    |   movel([0.647232, -1.413618, -2.553262, -0.745508, 1.570796, 2.218028],accel_mss,speed_ms,0,blend_radius_m)
    |   movel([0.645203, -1.414719, -2.552433, -0.745237, 1.570796, 2.216000],accel_mss,speed_ms,0,blend_radius_m)
    |   speed_ms = 0.005
    |   movel([0.645203, -1.406157, -2.548592, -0.757639, 1.570796, 2.216000],accel_mss,speed_ms,0,blend_radius_m)
    |   speed_ms = 0.040
    |   movel([0.644708, -1.402598, -2.551232, -0.758559, 1.570796, 2.215504],accel_mss,speed_ms,0,blend_radius_m)
    |   speed_ms = 0.005
    |   movel([0.644708, -1.411187, -2.555088, -0.746114, 1.570796, 2.215504],accel_mss,speed_ms,0,blend_radius_m)
    |   speed_ms = 0.025
    |   movel([0.632928, -1.420166, -2.548302, -0.743920, 1.570796, 2.203724],accel_mss,speed_ms,0,blend_radius_m)
    |   movel([0.632254, -1.420811, -2.547810, -0.743767, 1.570796, 2.203050],accel_mss,speed_ms,0,blend_radius_m)
    |   movel([0.631894, -1.421742, -2.547099, -0.743548, 1.570796, 2.202690],accel_mss,speed_ms,0,blend_radius_m)
    |   movel([0.631428, -1.422941, -2.546181, -0.743267, 1.570796, 2.202224],accel_mss,speed_ms,0,blend_radius_m)
    |   movel([0.630697, -1.424121, -2.545275, -0.742992, 1.570796, 2.201494],accel_mss,speed_ms,0,blend_radius_m)
    |   speed_ms = 0.005
    |   movel([0.630697, -1.415631, -2.541475, -0.755283, 1.570796, 2.201494],accel_mss,speed_ms,0,blend_radius_m)
    |   speed_ms = 0.040
    |   movel([0.643692, -1.414403, -2.542405, -0.755581, 1.570796, 2.214488],accel_mss,speed_ms,0,blend_radius_m)
    |   speed_ms = 0.005
    |   movel([0.643692, -1.422902, -2.546211, -0.743276, 1.570796, 2.214488],accel_mss,speed_ms,0,blend_radius_m)
    |   speed_ms = 0.025
    |   movel([0.644486, -1.421667, -2.547157, -0.743566, 1.570796, 2.215283],accel_mss,speed_ms,0,blend_radius_m)
    |   movel([0.645426, -1.420470, -2.548071, -0.743848, 1.570796, 2.216222],accel_mss,speed_ms,0,blend_radius_m)
    |   movel([0.646493, -1.419333, -2.548937, -0.744119, 1.570796, 2.217289],accel_mss,speed_ms,0,blend_radius_m)
    |   movel([0.647675, -1.418273, -2.549743, -0.744373, 1.570796, 2.218471],accel_mss,speed_ms,0,blend_radius_m)
    |   movel([0.648555, -1.417600, -2.550254, -0.744535, 1.570796, 2.219351],accel_mss,speed_ms,0,blend_radius_m)
    |   movel([0.649486, -1.417003, -2.550706, -0.744680, 1.570796, 2.220283],accel_mss,speed_ms,0,blend_radius_m)
    |   movel([0.650446, -1.416529, -2.551066, -0.744795, 1.570796, 2.221242],accel_mss,speed_ms,0,blend_radius_m)
    |   movel([0.651421, -1.416216, -2.551302, -0.744871, 1.570796, 2.222217],accel_mss,speed_ms,0,blend_radius_m)
    |   movel([0.652201, -1.416139, -2.551360, -0.744889, 1.570796, 2.222997],accel_mss,speed_ms,0,blend_radius_m)
    |   movel([0.652960, -1.416240, -2.551284, -0.744865, 1.570796, 2.223756],accel_mss,speed_ms,0,blend_radius_m)
    |   movel([0.653689, -1.416481, -2.551102, -0.744806, 1.570796, 2.224486],accel_mss,speed_ms,0,blend_radius_m)
    |   movel([0.654385, -1.416828, -2.550839, -0.744722, 1.570796, 2.225181],accel_mss,speed_ms,0,blend_radius_m)
    |   movel([0.655645, -1.417690, -2.550186, -0.744513, 1.570796, 2.226441],accel_mss,speed_ms,0,blend_radius_m)
    |   movel([0.656685, -1.418543, -2.549538, -0.744308, 1.570796, 2.227481],accel_mss,speed_ms,0,blend_radius_m)
    |   movel([0.655905, -1.418044, -2.549917, -0.744428, 1.570796, 2.226701],accel_mss,speed_ms,0,blend_radius_m)
    |   movel([0.654985, -1.417739, -2.550148, -0.744502, 1.570796, 2.225782],accel_mss,speed_ms,0,blend_radius_m)
    |   movel([0.653930, -1.417662, -2.550207, -0.744520, 1.570796, 2.224726],accel_mss,speed_ms,0,blend_radius_m)
    |   movel([0.652738, -1.417850, -2.550064, -0.744475, 1.570796, 2.223534],accel_mss,speed_ms,0,blend_radius_m)
    |   movel([0.651666, -1.418237, -2.549770, -0.744382, 1.570796, 2.222463],accel_mss,speed_ms,0,blend_radius_m)
    |   movel([0.650613, -1.418779, -2.549358, -0.744251, 1.570796, 2.221410],accel_mss,speed_ms,0,blend_radius_m)
    |   movel([0.649643, -1.419392, -2.548892, -0.744105, 1.570796, 2.220440],accel_mss,speed_ms,0,blend_radius_m)
    |   movel([0.648729, -1.420086, -2.548363, -0.743939, 1.570796, 2.219525],accel_mss,speed_ms,0,blend_radius_m)
    |   movel([0.647076, -1.421670, -2.547154, -0.743565, 1.570796, 2.217872],accel_mss,speed_ms,0,blend_radius_m)
    |   movel([0.645680, -1.423421, -2.545813, -0.743155, 1.570796, 2.216476],accel_mss,speed_ms,0,blend_radius_m)
    |   movel([0.644476, -1.425396, -2.544295, -0.742698, 1.570796, 2.215272],accel_mss,speed_ms,0,blend_radius_m)
    |   speed_ms = 0.005
    |   movel([0.644476, -1.416915, -2.540500, -0.754974, 1.570796, 2.215272],accel_mss,speed_ms,0,blend_radius_m)
    |   speed_ms = 0.040
    |   movel([0.649184, -1.413818, -2.542847, -0.755724, 1.570796, 2.219981],accel_mss,speed_ms,0,blend_radius_m)
    |   speed_ms = 0.005
    |   movel([0.649184, -1.422322, -2.546655, -0.743412, 1.570796, 2.219981],accel_mss,speed_ms,0,blend_radius_m)
    |   speed_ms = 0.025
    |   movel([0.648903, -1.422543, -2.546486, -0.743360, 1.570796, 2.219700],accel_mss,speed_ms,0,blend_radius_m)
    |   movel([0.648598, -1.422527, -2.546498, -0.743364, 1.570796, 2.219395],accel_mss,speed_ms,0,blend_radius_m)
    |   movel([0.648528, -1.422285, -2.546684, -0.743420, 1.570796, 2.219324],accel_mss,speed_ms,0,blend_radius_m)
    |   movel([0.648665, -1.421972, -2.546923, -0.743494, 1.570796, 2.219461],accel_mss,speed_ms,0,blend_radius_m)
    |   movel([0.649263, -1.421482, -2.547298, -0.743609, 1.570796, 2.220060],accel_mss,speed_ms,0,blend_radius_m)
    |   movel([0.649575, -1.421351, -2.547398, -0.743640, 1.570796, 2.220372],accel_mss,speed_ms,0,blend_radius_m)
    |   movel([0.649805, -1.421455, -2.547318, -0.743615, 1.570796, 2.220601],accel_mss,speed_ms,0,blend_radius_m)
    |   movel([0.649814, -1.421733, -2.547106, -0.743550, 1.570796, 2.220610],accel_mss,speed_ms,0,blend_radius_m)
    |   movel([0.649380, -1.422307, -2.546666, -0.743415, 1.570796, 2.220177],accel_mss,speed_ms,0,blend_radius_m)
    |   speed_ms = 0.005
    |   movel([0.649380, -1.413803, -2.542859, -0.755727, 1.570796, 2.220177],accel_mss,speed_ms,0,blend_radius_m)
    |   speed_ms = 0.040
    |   movel([0.644877, -1.421865, -2.536719, -0.753805, 1.570796, 2.215673],accel_mss,speed_ms,0,blend_radius_m)
    |   speed_ms = 0.005
    |   movel([0.644877, -1.430308, -2.540493, -0.741588, 1.570796, 2.215673],accel_mss,speed_ms,0,blend_radius_m)
    |   speed_ms = 0.025
    |   movel([0.646228, -1.429676, -2.540984, -0.741729, 1.570796, 2.217025],accel_mss,speed_ms,0,blend_radius_m)
    |   movel([0.647479, -1.428899, -2.541587, -0.741903, 1.570796, 2.218275],accel_mss,speed_ms,0,blend_radius_m)
    |   movel([0.649990, -1.427329, -2.542803, -0.742257, 1.570796, 2.220786],accel_mss,speed_ms,0,blend_radius_m)
    |   movel([0.651879, -1.426482, -2.543457, -0.742450, 1.570796, 2.222676],accel_mss,speed_ms,0,blend_radius_m)
    |   movel([0.657788, -1.424441, -2.545030, -0.742919, 1.570796, 2.228584],accel_mss,speed_ms,0,blend_radius_m)
    |   movel([0.658989, -1.423871, -2.545467, -0.743050, 1.570796, 2.229786],accel_mss,speed_ms,0,blend_radius_m)
    |   movel([0.659479, -1.423475, -2.545772, -0.743143, 1.570796, 2.230276],accel_mss,speed_ms,0,blend_radius_m)
    |   movel([0.659777, -1.422996, -2.546139, -0.743254, 1.570796, 2.230574],accel_mss,speed_ms,0,blend_radius_m)
    |   movel([0.659769, -1.422425, -2.546576, -0.743387, 1.570796, 2.230566],accel_mss,speed_ms,0,blend_radius_m)
    |   movel([0.659492, -1.421965, -2.546929, -0.743495, 1.570796, 2.230288],accel_mss,speed_ms,0,blend_radius_m)
    |   movel([0.658947, -1.421394, -2.547365, -0.743630, 1.570796, 2.229744],accel_mss,speed_ms,0,blend_radius_m)
    |   movel([0.658295, -1.421032, -2.547641, -0.743715, 1.570796, 2.229091],accel_mss,speed_ms,0,blend_radius_m)
    |   movel([0.657480, -1.420873, -2.547763, -0.743753, 1.570796, 2.228276],accel_mss,speed_ms,0,blend_radius_m)
    |   movel([0.656449, -1.420910, -2.547735, -0.743744, 1.570796, 2.227245],accel_mss,speed_ms,0,blend_radius_m)
    |   movel([0.655264, -1.421153, -2.547549, -0.743687, 1.570796, 2.226060],accel_mss,speed_ms,0,blend_radius_m)
    |   movel([0.654014, -1.421592, -2.547214, -0.743583, 1.570796, 2.224810],accel_mss,speed_ms,0,blend_radius_m)
    |   movel([0.652729, -1.422184, -2.546761, -0.743444, 1.570796, 2.223525],accel_mss,speed_ms,0,blend_radius_m)
    |   movel([0.651431, -1.422893, -2.546218, -0.743278, 1.570796, 2.222227],accel_mss,speed_ms,0,blend_radius_m)
    |   movel([0.648915, -1.424490, -2.544992, -0.742907, 1.570796, 2.219711],accel_mss,speed_ms,0,blend_radius_m)
    |   movel([0.646678, -1.426064, -2.543780, -0.742545, 1.570796, 2.217474],accel_mss,speed_ms,0,blend_radius_m)
    |   movel([0.642614, -1.429086, -2.541442, -0.741861, 1.570796, 2.213410],accel_mss,speed_ms,0,blend_radius_m)
    |   movel([0.641217, -1.430012, -2.540723, -0.741654, 1.570796, 2.212013],accel_mss,speed_ms,0,blend_radius_m)
    |   movel([0.639755, -1.430829, -2.540087, -0.741473, 1.570796, 2.210551],accel_mss,speed_ms,0,blend_radius_m)
    |   movel([0.638252, -1.431473, -2.539586, -0.741330, 1.570796, 2.209049],accel_mss,speed_ms,0,blend_radius_m)
    |   movel([0.636769, -1.431875, -2.539272, -0.741242, 1.570796, 2.207566],accel_mss,speed_ms,0,blend_radius_m)
    |   movel([0.635365, -1.431969, -2.539199, -0.741221, 1.570796, 2.206162],accel_mss,speed_ms,0,blend_radius_m)
    |   movel([0.636219, -1.432324, -2.538922, -0.741143, 1.570796, 2.207016],accel_mss,speed_ms,0,blend_radius_m)
    |   movel([0.637153, -1.432573, -2.538727, -0.741089, 1.570796, 2.207950],accel_mss,speed_ms,0,blend_radius_m)
    |   movel([0.638159, -1.432712, -2.538619, -0.741058, 1.570796, 2.208955],accel_mss,speed_ms,0,blend_radius_m)
    |   movel([0.639218, -1.432740, -2.538596, -0.741052, 1.570796, 2.210014],accel_mss,speed_ms,0,blend_radius_m)
    |   movel([0.638520, -1.433919, -2.537675, -0.740796, 1.570796, 2.209316],accel_mss,speed_ms,0,blend_radius_m)
    |   movel([0.637653, -1.435054, -2.536785, -0.740551, 1.570796, 2.208449],accel_mss,speed_ms,0,blend_radius_m)
    |   movel([0.636642, -1.436119, -2.535948, -0.740322, 1.570796, 2.207438],accel_mss,speed_ms,0,blend_radius_m)
    |   movel([0.635508, -1.437089, -2.535184, -0.740116, 1.570796, 2.206304],accel_mss,speed_ms,0,blend_radius_m)
    |   movel([0.637021, -1.436449, -2.535688, -0.740252, 1.570796, 2.207818],accel_mss,speed_ms,0,blend_radius_m)
    |   movel([0.638475, -1.435651, -2.536316, -0.740422, 1.570796, 2.209271],accel_mss,speed_ms,0,blend_radius_m)
    |   movel([0.639868, -1.434716, -2.537050, -0.740623, 1.570796, 2.210664],accel_mss,speed_ms,0,blend_radius_m)
    |   movel([0.641204, -1.433667, -2.537872, -0.740850, 1.570796, 2.212000],accel_mss,speed_ms,0,blend_radius_m)
    |   movel([0.640775, -1.434467, -2.537245, -0.740677, 1.570796, 2.211571],accel_mss,speed_ms,0,blend_radius_m)
    |   movel([0.640145, -1.435303, -2.536589, -0.740497, 1.570796, 2.210942],accel_mss,speed_ms,0,blend_radius_m)
    |   movel([0.636793, -1.438812, -2.533824, -0.739753, 1.570796, 2.207590],accel_mss,speed_ms,0,blend_radius_m)
    |   movel([0.636040, -1.439697, -2.533123, -0.739568, 1.570796, 2.206837],accel_mss,speed_ms,0,blend_radius_m)
    |   movel([0.635442, -1.440567, -2.532434, -0.739388, 1.570796, 2.206238],accel_mss,speed_ms,0,blend_radius_m)
    |   movel([0.636724, -1.439441, -2.533327, -0.739622, 1.570796, 2.207520],accel_mss,speed_ms,0,blend_radius_m)
    |   movel([0.638005, -1.438470, -2.534094, -0.739825, 1.570796, 2.208801],accel_mss,speed_ms,0,blend_radius_m)
    |   movel([0.640578, -1.436842, -2.535379, -0.740168, 1.570796, 2.211374],accel_mss,speed_ms,0,blend_radius_m)
    |   movel([0.643201, -1.435348, -2.536554, -0.740487, 1.570796, 2.213998],accel_mss,speed_ms,0,blend_radius_m)
    |   movel([0.645926, -1.433653, -2.537883, -0.740853, 1.570796, 2.216722],accel_mss,speed_ms,0,blend_radius_m)
    |   movel([0.647510, -1.432448, -2.538825, -0.741116, 1.570796, 2.218306],accel_mss,speed_ms,0,blend_radius_m)
    |   movel([0.648453, -1.431852, -2.539290, -0.741247, 1.570796, 2.219250],accel_mss,speed_ms,0,blend_radius_m)
    |   movel([0.648851, -1.431691, -2.539416, -0.741282, 1.570796, 2.219647],accel_mss,speed_ms,0,blend_radius_m)
    |   movel([0.649160, -1.431671, -2.539432, -0.741287, 1.570796, 2.219957],accel_mss,speed_ms,0,blend_radius_m)
    |   movel([0.649355, -1.431804, -2.539328, -0.741258, 1.570796, 2.220151],accel_mss,speed_ms,0,blend_radius_m)
    |   movel([0.649443, -1.432056, -2.539131, -0.741202, 1.570796, 2.220239],accel_mss,speed_ms,0,blend_radius_m)
    |   movel([0.649367, -1.432776, -2.538568, -0.741044, 1.570796, 2.220164],accel_mss,speed_ms,0,blend_radius_m)
    |   movel([0.649054, -1.433558, -2.537957, -0.740874, 1.570796, 2.219850],accel_mss,speed_ms,0,blend_radius_m)
    |   movel([0.648620, -1.434127, -2.537512, -0.740751, 1.570796, 2.219417],accel_mss,speed_ms,0,blend_radius_m)
    |   movel([0.650492, -1.432463, -2.538813, -0.741113, 1.570796, 2.221288],accel_mss,speed_ms,0,blend_radius_m)
    |   movel([0.652210, -1.430675, -2.540207, -0.741507, 1.570796, 2.223006],accel_mss,speed_ms,0,blend_radius_m)
    |   movel([0.653753, -1.428790, -2.541671, -0.741927, 1.570796, 2.224549],accel_mss,speed_ms,0,blend_radius_m)
    |   movel([0.655098, -1.426832, -2.543187, -0.742370, 1.570796, 2.225894],accel_mss,speed_ms,0,blend_radius_m)
    |   speed_ms = 0.005
    |   movel([0.655098, -1.418363, -2.539398, -0.754628, 1.570796, 2.225894],accel_mss,speed_ms,0,blend_radius_m)
    |   speed_ms = 0.040
    |   movel([0.656273, -1.420049, -2.538111, -0.754229, 1.570796, 2.227069],accel_mss,speed_ms,0,blend_radius_m)
    |   speed_ms = 0.005
    |   movel([0.656273, -1.428505, -2.541892, -0.741991, 1.570796, 2.227069],accel_mss,speed_ms,0,blend_radius_m)
    |   speed_ms = 0.025
    |   movel([0.657037, -1.429367, -2.541224, -0.741798, 1.570796, 2.227833],accel_mss,speed_ms,0,blend_radius_m)
    |   movel([0.657209, -1.429905, -2.540806, -0.741678, 1.570796, 2.228005],accel_mss,speed_ms,0,blend_radius_m)
    |   movel([0.657126, -1.430531, -2.540319, -0.741539, 1.570796, 2.227923],accel_mss,speed_ms,0,blend_radius_m)
    |   movel([0.656831, -1.431094, -2.539881, -0.741414, 1.570796, 2.227628],accel_mss,speed_ms,0,blend_radius_m)
    |   movel([0.650125, -1.439891, -2.532970, -0.739528, 1.570796, 2.220921],accel_mss,speed_ms,0,blend_radius_m)
    |   movel([0.649615, -1.440501, -2.532486, -0.739402, 1.570796, 2.220412],accel_mss,speed_ms,0,blend_radius_m)
    |   movel([0.649027, -1.441062, -2.532041, -0.739286, 1.570796, 2.219823],accel_mss,speed_ms,0,blend_radius_m)
    |   movel([0.648392, -1.441459, -2.531726, -0.739204, 1.570796, 2.219189],accel_mss,speed_ms,0,blend_radius_m)
    |   movel([0.647752, -1.441583, -2.531627, -0.739179, 1.570796, 2.218548],accel_mss,speed_ms,0,blend_radius_m)
    |   movel([0.647286, -1.441405, -2.531769, -0.739215, 1.570796, 2.218082],accel_mss,speed_ms,0,blend_radius_m)
    |   movel([0.646586, -1.440749, -2.532289, -0.739350, 1.570796, 2.217382],accel_mss,speed_ms,0,blend_radius_m)
    |   movel([0.646108, -1.440597, -2.532410, -0.739382, 1.570796, 2.216904],accel_mss,speed_ms,0,blend_radius_m)
    |   movel([0.645368, -1.440782, -2.532264, -0.739344, 1.570796, 2.216164],accel_mss,speed_ms,0,blend_radius_m)
    |   movel([0.644608, -1.441155, -2.531967, -0.739267, 1.570796, 2.215405],accel_mss,speed_ms,0,blend_radius_m)
    |   movel([0.643699, -1.441518, -2.531678, -0.739192, 1.570796, 2.214496],accel_mss,speed_ms,0,blend_radius_m)
    |   movel([0.642798, -1.441723, -2.531515, -0.739150, 1.570796, 2.213595],accel_mss,speed_ms,0,blend_radius_m)
    |   movel([0.641935, -1.441776, -2.531473, -0.739139, 1.570796, 2.212731],accel_mss,speed_ms,0,blend_radius_m)
    |   movel([0.641134, -1.441682, -2.531548, -0.739159, 1.570796, 2.211931],accel_mss,speed_ms,0,blend_radius_m)
    |   movel([0.640423, -1.441448, -2.531735, -0.739207, 1.570796, 2.211219],accel_mss,speed_ms,0,blend_radius_m)
    |   movel([0.639832, -1.441078, -2.532029, -0.739283, 1.570796, 2.210629],accel_mss,speed_ms,0,blend_radius_m)
    |   movel([0.639385, -1.440582, -2.532422, -0.739385, 1.570796, 2.210182],accel_mss,speed_ms,0,blend_radius_m)
    |   movel([0.639114, -1.439959, -2.532916, -0.739514, 1.570796, 2.209910],accel_mss,speed_ms,0,blend_radius_m)
    |   speed_ms = 0.005
    |   movel([0.639114, -1.431591, -2.529183, -0.751615, 1.570796, 2.209910],accel_mss,speed_ms,0,blend_radius_m)
    |   speed_ms = 0.040
    |   movel([0.629566, -1.437668, -2.524402, -0.750318, 1.570796, 2.200362],accel_mss,speed_ms,0,blend_radius_m)
    |   speed_ms = 0.005
    |   movel([0.629566, -1.445989, -2.528110, -0.738290, 1.570796, 2.200362],accel_mss,speed_ms,0,blend_radius_m)
    |   speed_ms = 0.025
    |   movel([0.624482, -1.455129, -2.520718, -0.736542, 1.570796, 2.195278],accel_mss,speed_ms,0,blend_radius_m)
    |   movel([0.623759, -1.456220, -2.519827, -0.736342, 1.570796, 2.194556],accel_mss,speed_ms,0,blend_radius_m)
    |   movel([0.623285, -1.456679, -2.519452, -0.736258, 1.570796, 2.194081],accel_mss,speed_ms,0,blend_radius_m)
    |   movel([0.622719, -1.457000, -2.519189, -0.736200, 1.570796, 2.193515],accel_mss,speed_ms,0,blend_radius_m)
    |   movel([0.621425, -1.457352, -2.518901, -0.736136, 1.570796, 2.192221],accel_mss,speed_ms,0,blend_radius_m)
    |   movel([0.620864, -1.457799, -2.518534, -0.736056, 1.570796, 2.191661],accel_mss,speed_ms,0,blend_radius_m)
    |   movel([0.620463, -1.458373, -2.518064, -0.735953, 1.570796, 2.191259],accel_mss,speed_ms,0,blend_radius_m)
    |   movel([0.620070, -1.459371, -2.517243, -0.735774, 1.570796, 2.190867],accel_mss,speed_ms,0,blend_radius_m)
    |   movel([0.619927, -1.460382, -2.516412, -0.735596, 1.570796, 2.190723],accel_mss,speed_ms,0,blend_radius_m)
    |   movel([0.619862, -1.462310, -2.514820, -0.735259, 1.570796, 2.190659],accel_mss,speed_ms,0,blend_radius_m)
    |   movel([0.619585, -1.463630, -2.513727, -0.735032, 1.570796, 2.190381],accel_mss,speed_ms,0,blend_radius_m)
    |   movel([0.618938, -1.465519, -2.512159, -0.734712, 1.570796, 2.189734],accel_mss,speed_ms,0,blend_radius_m)
    |   movel([0.618503, -1.466353, -2.511464, -0.734572, 1.570796, 2.189299],accel_mss,speed_ms,0,blend_radius_m)
    |   movel([0.618001, -1.466949, -2.510967, -0.734473, 1.570796, 2.188798],accel_mss,speed_ms,0,blend_radius_m)
    |   movel([0.617730, -1.467114, -2.510829, -0.734446, 1.570796, 2.188526],accel_mss,speed_ms,0,blend_radius_m)
    |   movel([0.617446, -1.467173, -2.510780, -0.734436, 1.570796, 2.188242],accel_mss,speed_ms,0,blend_radius_m)
    |   movel([0.617150, -1.467109, -2.510834, -0.734446, 1.570796, 2.187946],accel_mss,speed_ms,0,blend_radius_m)
    |   movel([0.616845, -1.466904, -2.511005, -0.734480, 1.570796, 2.187641],accel_mss,speed_ms,0,blend_radius_m)
    |   movel([0.616369, -1.467578, -2.510442, -0.734369, 1.570796, 2.187165],accel_mss,speed_ms,0,blend_radius_m)
    |   movel([0.616008, -1.468390, -2.509763, -0.734236, 1.570796, 2.186804],accel_mss,speed_ms,0,blend_radius_m)
    |   movel([0.615555, -1.470239, -2.508214, -0.733936, 1.570796, 2.186351],accel_mss,speed_ms,0,blend_radius_m)
    |   movel([0.615357, -1.472073, -2.506672, -0.733644, 1.570796, 2.186154],accel_mss,speed_ms,0,blend_radius_m)
    |   movel([0.615291, -1.473520, -2.505452, -0.733417, 1.570796, 2.186088],accel_mss,speed_ms,0,blend_radius_m)
    |   movel([0.615441, -1.475063, -2.504147, -0.733179, 1.570796, 2.186237],accel_mss,speed_ms,0,blend_radius_m)
    |   movel([0.615759, -1.476614, -2.502832, -0.732943, 1.570796, 2.186556],accel_mss,speed_ms,0,blend_radius_m)
    |   movel([0.615875, -1.478202, -2.501481, -0.732706, 1.570796, 2.186672],accel_mss,speed_ms,0,blend_radius_m)
    |   movel([0.615743, -1.479016, -2.500787, -0.732586, 1.570796, 2.186540],accel_mss,speed_ms,0,blend_radius_m)
    |   movel([0.615421, -1.479850, -2.500076, -0.732464, 1.570796, 2.186217],accel_mss,speed_ms,0,blend_radius_m)
    |   movel([0.615143, -1.480267, -2.499719, -0.732403, 1.570796, 2.185940],accel_mss,speed_ms,0,blend_radius_m)
    |   movel([0.614767, -1.480641, -2.499399, -0.732349, 1.570796, 2.185563],accel_mss,speed_ms,0,blend_radius_m)
    |   movel([0.614354, -1.480878, -2.499196, -0.732315, 1.570796, 2.185150],accel_mss,speed_ms,0,blend_radius_m)
    |   movel([0.613964, -1.480890, -2.499186, -0.732313, 1.570796, 2.184760],accel_mss,speed_ms,0,blend_radius_m)
    |   movel([0.613760, -1.480715, -2.499336, -0.732338, 1.570796, 2.184557],accel_mss,speed_ms,0,blend_radius_m)
    |   movel([0.613656, -1.480463, -2.499551, -0.732375, 1.570796, 2.184453],accel_mss,speed_ms,0,blend_radius_m)
    |   movel([0.613063, -1.477851, -2.501780, -0.732758, 1.570796, 2.183860],accel_mss,speed_ms,0,blend_radius_m)
    |   movel([0.612918, -1.476478, -2.502947, -0.732964, 1.570796, 2.183714],accel_mss,speed_ms,0,blend_radius_m)
    |   movel([0.612878, -1.475065, -2.504146, -0.733178, 1.570796, 2.183674],accel_mss,speed_ms,0,blend_radius_m)
    |   movel([0.612419, -1.475366, -2.503891, -0.733132, 1.570796, 2.183216],accel_mss,speed_ms,0,blend_radius_m)
    |   movel([0.612028, -1.475740, -2.503573, -0.733075, 1.570796, 2.182824],accel_mss,speed_ms,0,blend_radius_m)
    |   movel([0.611430, -1.476666, -2.502787, -0.732935, 1.570796, 2.182227],accel_mss,speed_ms,0,blend_radius_m)
    |   movel([0.611042, -1.477762, -2.501856, -0.732771, 1.570796, 2.181838],accel_mss,speed_ms,0,blend_radius_m)
    |   movel([0.610826, -1.478948, -2.500845, -0.732596, 1.570796, 2.181622],accel_mss,speed_ms,0,blend_radius_m)
    |   movel([0.610731, -1.481288, -2.498845, -0.732256, 1.570796, 2.181528],accel_mss,speed_ms,0,blend_radius_m)
    |   movel([0.610820, -1.483067, -2.497319, -0.732003, 1.570796, 2.181616],accel_mss,speed_ms,0,blend_radius_m)
    |   movel([0.610778, -1.483746, -2.496735, -0.731908, 1.570796, 2.181574],accel_mss,speed_ms,0,blend_radius_m)
    |   movel([0.610645, -1.484082, -2.496446, -0.731861, 1.570796, 2.181441],accel_mss,speed_ms,0,blend_radius_m)
    |   movel([0.610384, -1.484388, -2.496182, -0.731819, 1.570796, 2.181181],accel_mss,speed_ms,0,blend_radius_m)
    |   movel([0.610011, -1.484627, -2.495976, -0.731786, 1.570796, 2.180807],accel_mss,speed_ms,0,blend_radius_m)
    |   movel([0.609698, -1.484694, -2.495918, -0.731777, 1.570796, 2.180495],accel_mss,speed_ms,0,blend_radius_m)
    |   movel([0.609210, -1.484500, -2.496086, -0.731803, 1.570796, 2.180006],accel_mss,speed_ms,0,blend_radius_m)
    |   movel([0.608588, -1.484138, -2.496398, -0.731854, 1.570796, 2.179384],accel_mss,speed_ms,0,blend_radius_m)
    |   movel([0.608354, -1.484199, -2.496345, -0.731845, 1.570796, 2.179151],accel_mss,speed_ms,0,blend_radius_m)
    |   movel([0.608059, -1.484440, -2.496137, -0.731812, 1.570796, 2.178855],accel_mss,speed_ms,0,blend_radius_m)
    |   movel([0.607831, -1.484776, -2.495847, -0.731765, 1.570796, 2.178627],accel_mss,speed_ms,0,blend_radius_m)
    |   movel([0.607540, -1.485617, -2.495122, -0.731650, 1.570796, 2.178336],accel_mss,speed_ms,0,blend_radius_m)
    |   movel([0.607317, -1.487165, -2.493784, -0.731441, 1.570796, 2.178114],accel_mss,speed_ms,0,blend_radius_m)
    |   movel([0.607067, -1.490393, -2.490980, -0.731016, 1.570796, 2.177864],accel_mss,speed_ms,0,blend_radius_m)
    |   movel([0.606894, -1.493587, -2.488190, -0.730612, 1.570796, 2.177690],accel_mss,speed_ms,0,blend_radius_m)
    |   movel([0.606763, -1.494250, -2.487609, -0.730530, 1.570796, 2.177559],accel_mss,speed_ms,0,blend_radius_m)
    |   movel([0.606487, -1.494923, -2.487018, -0.730448, 1.570796, 2.177283],accel_mss,speed_ms,0,blend_radius_m)
    |   movel([0.606041, -1.495494, -2.486517, -0.730379, 1.570796, 2.176838],accel_mss,speed_ms,0,blend_radius_m)
    |   movel([0.605751, -1.495705, -2.486331, -0.730353, 1.570796, 2.176547],accel_mss,speed_ms,0,blend_radius_m)
    |   movel([0.605086, -1.495899, -2.486161, -0.730330, 1.570796, 2.175882],accel_mss,speed_ms,0,blend_radius_m)
    |   movel([0.604813, -1.495863, -2.486192, -0.730334, 1.570796, 2.175609],accel_mss,speed_ms,0,blend_radius_m)
    |   movel([0.604396, -1.495580, -2.486441, -0.730368, 1.570796, 2.175192],accel_mss,speed_ms,0,blend_radius_m)
    |   movel([0.604131, -1.495116, -2.486849, -0.730424, 1.570796, 2.174927],accel_mss,speed_ms,0,blend_radius_m)
    |   movel([0.603992, -1.494579, -2.487320, -0.730490, 1.570796, 2.174788],accel_mss,speed_ms,0,blend_radius_m)
    |   movel([0.603563, -1.491248, -2.490235, -0.730906, 1.570796, 2.174360],accel_mss,speed_ms,0,blend_radius_m)
    |   movel([0.603337, -1.487825, -2.493211, -0.731352, 1.570796, 2.174133],accel_mss,speed_ms,0,blend_radius_m)
    |   movel([0.603320, -1.484316, -2.496244, -0.731829, 1.570796, 2.174117],accel_mss,speed_ms,0,blend_radius_m)
    |   movel([0.603515, -1.480728, -2.499325, -0.732336, 1.570796, 2.174312],accel_mss,speed_ms,0,blend_radius_m)
    |   movel([0.603673, -1.479373, -2.500483, -0.732533, 1.570796, 2.174470],accel_mss,speed_ms,0,blend_radius_m)
    |   movel([0.604054, -1.477986, -2.501666, -0.732738, 1.570796, 2.174850],accel_mss,speed_ms,0,blend_radius_m)
    |   movel([0.604445, -1.477158, -2.502370, -0.732861, 1.570796, 2.175241],accel_mss,speed_ms,0,blend_radius_m)
    |   movel([0.604935, -1.476340, -2.503064, -0.732984, 1.570796, 2.175732],accel_mss,speed_ms,0,blend_radius_m)
    |   movel([0.606078, -1.474727, -2.504431, -0.733230, 1.570796, 2.176875],accel_mss,speed_ms,0,blend_radius_m)
    |   movel([0.610693, -1.469097, -2.509172, -0.734120, 1.570796, 2.181490],accel_mss,speed_ms,0,blend_radius_m)
    |   movel([0.611871, -1.467453, -2.510546, -0.734389, 1.570796, 2.182668],accel_mss,speed_ms,0,blend_radius_m)
    |   movel([0.612764, -1.465916, -2.511828, -0.734645, 1.570796, 2.183560],accel_mss,speed_ms,0,blend_radius_m)
    |   movel([0.613060, -1.465219, -2.512408, -0.734762, 1.570796, 2.183856],accel_mss,speed_ms,0,blend_radius_m)
    |   movel([0.613226, -1.464587, -2.512933, -0.734869, 1.570796, 2.184023],accel_mss,speed_ms,0,blend_radius_m)
    |   movel([0.613249, -1.464033, -2.513393, -0.734963, 1.570796, 2.184045],accel_mss,speed_ms,0,blend_radius_m)
    |   movel([0.613109, -1.463570, -2.513777, -0.735042, 1.570796, 2.183906],accel_mss,speed_ms,0,blend_radius_m)
    |   movel([0.612615, -1.462930, -2.514307, -0.735152, 1.570796, 2.183411],accel_mss,speed_ms,0,blend_radius_m)
    |   movel([0.612428, -1.462587, -2.514591, -0.735211, 1.570796, 2.183224],accel_mss,speed_ms,0,blend_radius_m)
    |   movel([0.612411, -1.462174, -2.514932, -0.735283, 1.570796, 2.183207],accel_mss,speed_ms,0,blend_radius_m)
    |   movel([0.612772, -1.461510, -2.515481, -0.735398, 1.570796, 2.183569],accel_mss,speed_ms,0,blend_radius_m)
    |   movel([0.613381, -1.460896, -2.515988, -0.735505, 1.570796, 2.184177],accel_mss,speed_ms,0,blend_radius_m)
    |   movel([0.615399, -1.458974, -2.517570, -0.735845, 1.570796, 2.186195],accel_mss,speed_ms,0,blend_radius_m)
    |   movel([0.617306, -1.456995, -2.519193, -0.736201, 1.570796, 2.188103],accel_mss,speed_ms,0,blend_radius_m)
    |   movel([0.619122, -1.454960, -2.520856, -0.736573, 1.570796, 2.189918],accel_mss,speed_ms,0,blend_radius_m)
    |   movel([0.620860, -1.452875, -2.522553, -0.736961, 1.570796, 2.191657],accel_mss,speed_ms,0,blend_radius_m)
    |   movel([0.624183, -1.448586, -2.526023, -0.737780, 1.570796, 2.194980],accel_mss,speed_ms,0,blend_radius_m)
    |   movel([0.627417, -1.444166, -2.529568, -0.738654, 1.570796, 2.198213],accel_mss,speed_ms,0,blend_radius_m)
    |   speed_ms = 0.005
    |   movel([0.627417, -1.435831, -2.525853, -0.750704, 1.570796, 2.198213],accel_mss,speed_ms,0,blend_radius_m)
    |   speed_ms = 0.040
    |   movel([0.617703, -1.446063, -2.517707, -0.748620, 1.570796, 2.188499],accel_mss,speed_ms,0,blend_radius_m)
    |   speed_ms = 0.005
    |   movel([0.617703, -1.454317, -2.521380, -0.736692, 1.570796, 2.188499],accel_mss,speed_ms,0,blend_radius_m)
    |   speed_ms = 0.025
    |   movel([0.614220, -1.456040, -2.519974, -0.736375, 1.570796, 2.185017],accel_mss,speed_ms,0,blend_radius_m)
    |   movel([0.610716, -1.457622, -2.518679, -0.736087, 1.570796, 2.181513],accel_mss,speed_ms,0,blend_radius_m)
    |   movel([0.607196, -1.459065, -2.517495, -0.735829, 1.570796, 2.177992],accel_mss,speed_ms,0,blend_radius_m)
    |   movel([0.603671, -1.460362, -2.516428, -0.735599, 1.570796, 2.174468],accel_mss,speed_ms,0,blend_radius_m)
    |   movel([0.606791, -1.458463, -2.517990, -0.735936, 1.570796, 2.177587],accel_mss,speed_ms,0,blend_radius_m)
    |   movel([0.609822, -1.456386, -2.519691, -0.736312, 1.570796, 2.180619],accel_mss,speed_ms,0,blend_radius_m)
    |   movel([0.612746, -1.454144, -2.521521, -0.736724, 1.570796, 2.183542],accel_mss,speed_ms,0,blend_radius_m)
    |   movel([0.615543, -1.451749, -2.523466, -0.737173, 1.570796, 2.186340],accel_mss,speed_ms,0,blend_radius_m)
    |   movel([0.612639, -1.453118, -2.522356, -0.736916, 1.570796, 2.183435],accel_mss,speed_ms,0,blend_radius_m)
    |   movel([0.609722, -1.454378, -2.521330, -0.736681, 1.570796, 2.180518],accel_mss,speed_ms,0,blend_radius_m)
    |   movel([0.606793, -1.455529, -2.520391, -0.736468, 1.570796, 2.177589],accel_mss,speed_ms,0,blend_radius_m)
    |   movel([0.603861, -1.456566, -2.519544, -0.736279, 1.570796, 2.174657],accel_mss,speed_ms,0,blend_radius_m)
    |   movel([0.600601, -1.457644, -2.518662, -0.736084, 1.570796, 2.171397],accel_mss,speed_ms,0,blend_radius_m)
    |   movel([0.597364, -1.458897, -2.517633, -0.735859, 1.570796, 2.168160],accel_mss,speed_ms,0,blend_radius_m)
    |   movel([0.595768, -1.459689, -2.516982, -0.735718, 1.570796, 2.166565],accel_mss,speed_ms,0,blend_radius_m)
    |   movel([0.594229, -1.460623, -2.516212, -0.735553, 1.570796, 2.165025],accel_mss,speed_ms,0,blend_radius_m)
    |   movel([0.592805, -1.461704, -2.515321, -0.735364, 1.570796, 2.163602],accel_mss,speed_ms,0,blend_radius_m)
    |   movel([0.591552, -1.462929, -2.514307, -0.735152, 1.570796, 2.162348],accel_mss,speed_ms,0,blend_radius_m)
    |   movel([0.592804, -1.461262, -2.515686, -0.735441, 1.570796, 2.163600],accel_mss,speed_ms,0,blend_radius_m)
    |   movel([0.594211, -1.459598, -2.517057, -0.735734, 1.570796, 2.165007],accel_mss,speed_ms,0,blend_radius_m)
    |   movel([0.595752, -1.457957, -2.518405, -0.736027, 1.570796, 2.166548],accel_mss,speed_ms,0,blend_radius_m)
    |   movel([0.597405, -1.456357, -2.519715, -0.736317, 1.570796, 2.168201],accel_mss,speed_ms,0,blend_radius_m)
    |   movel([0.599146, -1.454818, -2.520971, -0.736599, 1.570796, 2.169942],accel_mss,speed_ms,0,blend_radius_m)
    |   movel([0.600954, -1.453361, -2.522158, -0.736870, 1.570796, 2.171750],accel_mss,speed_ms,0,blend_radius_m)
    |   movel([0.602805, -1.452004, -2.523260, -0.737125, 1.570796, 2.173601],accel_mss,speed_ms,0,blend_radius_m)
    |   movel([0.604675, -1.450769, -2.524260, -0.737360, 1.570796, 2.175471],accel_mss,speed_ms,0,blend_radius_m)
    |   movel([0.601533, -1.452451, -2.522897, -0.737041, 1.570796, 2.172329],accel_mss,speed_ms,0,blend_radius_m)
    |   movel([0.598460, -1.454267, -2.521421, -0.736701, 1.570796, 2.169257],accel_mss,speed_ms,0,blend_radius_m)
    |   movel([0.595458, -1.456198, -2.519845, -0.736346, 1.570796, 2.166254],accel_mss,speed_ms,0,blend_radius_m)
    |   movel([0.592526, -1.458228, -2.518182, -0.735978, 1.570796, 2.163322],accel_mss,speed_ms,0,blend_radius_m)
    |   movel([0.589668, -1.460337, -2.516448, -0.735603, 1.570796, 2.160464],accel_mss,speed_ms,0,blend_radius_m)
    |   movel([0.586882, -1.462508, -2.514656, -0.735225, 1.570796, 2.157678],accel_mss,speed_ms,0,blend_radius_m)
    |   movel([0.581527, -1.466961, -2.510957, -0.734471, 1.570796, 2.152324],accel_mss,speed_ms,0,blend_radius_m)
    |   movel([0.583200, -1.465285, -2.512353, -0.734751, 1.570796, 2.153996],accel_mss,speed_ms,0,blend_radius_m)
    |   movel([0.584790, -1.463356, -2.513954, -0.735079, 1.570796, 2.155586],accel_mss,speed_ms,0,blend_radius_m)
    |   movel([0.587772, -1.459527, -2.517115, -0.735747, 1.570796, 2.158569],accel_mss,speed_ms,0,blend_radius_m)
    |   movel([0.589223, -1.457899, -2.518453, -0.736038, 1.570796, 2.160019],accel_mss,speed_ms,0,blend_radius_m)
    |   movel([0.590627, -1.456498, -2.519600, -0.736291, 1.570796, 2.161423],accel_mss,speed_ms,0,blend_radius_m)
    |   movel([0.593740, -1.453771, -2.521825, -0.736794, 1.570796, 2.164536],accel_mss,speed_ms,0,blend_radius_m)
    |   movel([0.593201, -1.454066, -2.521585, -0.736739, 1.570796, 2.163998],accel_mss,speed_ms,0,blend_radius_m)
    |   movel([0.592392, -1.454326, -2.521373, -0.736690, 1.570796, 2.163188],accel_mss,speed_ms,0,blend_radius_m)
    |   movel([0.588113, -1.455156, -2.520696, -0.736537, 1.570796, 2.158910],accel_mss,speed_ms,0,blend_radius_m)
    |   movel([0.586531, -1.455538, -2.520385, -0.736467, 1.570796, 2.157327],accel_mss,speed_ms,0,blend_radius_m)
    |   movel([0.584569, -1.456412, -2.519671, -0.736307, 1.570796, 2.155365],accel_mss,speed_ms,0,blend_radius_m)
    |   movel([0.582619, -1.457507, -2.518774, -0.736108, 1.570796, 2.153415],accel_mss,speed_ms,0,blend_radius_m)
    |   movel([0.578875, -1.459968, -2.516752, -0.735669, 1.570796, 2.149671],accel_mss,speed_ms,0,blend_radius_m)
    |   movel([0.580598, -1.458430, -2.518017, -0.735942, 1.570796, 2.151394],accel_mss,speed_ms,0,blend_radius_m)
    |   movel([0.582217, -1.456797, -2.519355, -0.736237, 1.570796, 2.153013],accel_mss,speed_ms,0,blend_radius_m)
    |   movel([0.585431, -1.453485, -2.522057, -0.736847, 1.570796, 2.156227],accel_mss,speed_ms,0,blend_radius_m)
    |   movel([0.587232, -1.451864, -2.523373, -0.737152, 1.570796, 2.158029],accel_mss,speed_ms,0,blend_radius_m)
    |   movel([0.589151, -1.450323, -2.524621, -0.737445, 1.570796, 2.159948],accel_mss,speed_ms,0,blend_radius_m)
    |   movel([0.593248, -1.447424, -2.526958, -0.738007, 1.570796, 2.164045],accel_mss,speed_ms,0,blend_radius_m)
    |   movel([0.601686, -1.442016, -2.531283, -0.739090, 1.570796, 2.172482],accel_mss,speed_ms,0,blend_radius_m)
    |   movel([0.599268, -1.442212, -2.531127, -0.739050, 1.570796, 2.170065],accel_mss,speed_ms,0,blend_radius_m)
    |   movel([0.596800, -1.442588, -2.530827, -0.738974, 1.570796, 2.167597],accel_mss,speed_ms,0,blend_radius_m)
    |   movel([0.594296, -1.443134, -2.530392, -0.738863, 1.570796, 2.165092],accel_mss,speed_ms,0,blend_radius_m)
    |   movel([0.591774, -1.443847, -2.529824, -0.738719, 1.570796, 2.162570],accel_mss,speed_ms,0,blend_radius_m)
    |   movel([0.589252, -1.444721, -2.529125, -0.738543, 1.570796, 2.160048],accel_mss,speed_ms,0,blend_radius_m)
    |   movel([0.586742, -1.445753, -2.528299, -0.738337, 1.570796, 2.157539],accel_mss,speed_ms,0,blend_radius_m)
    |   movel([0.584263, -1.446932, -2.527353, -0.738104, 1.570796, 2.155060],accel_mss,speed_ms,0,blend_radius_m)
    |   movel([0.581830, -1.448255, -2.526289, -0.737845, 1.570796, 2.152627],accel_mss,speed_ms,0,blend_radius_m)
    |   movel([0.582525, -1.447792, -2.526662, -0.737935, 1.570796, 2.153321],accel_mss,speed_ms,0,blend_radius_m)
    |   movel([0.583240, -1.447212, -2.527128, -0.738049, 1.570796, 2.154036],accel_mss,speed_ms,0,blend_radius_m)
    |   movel([0.584694, -1.445834, -2.528234, -0.738321, 1.570796, 2.155491],accel_mss,speed_ms,0,blend_radius_m)
    |   movel([0.587424, -1.443136, -2.530391, -0.738862, 1.570796, 2.158220],accel_mss,speed_ms,0,blend_radius_m)
    |   movel([0.589964, -1.441002, -2.532089, -0.739298, 1.570796, 2.160760],accel_mss,speed_ms,0,blend_radius_m)
    |   movel([0.592572, -1.438953, -2.533713, -0.739724, 1.570796, 2.163369],accel_mss,speed_ms,0,blend_radius_m)
    |   movel([0.595245, -1.436986, -2.535265, -0.740138, 1.570796, 2.166041],accel_mss,speed_ms,0,blend_radius_m)
    |   movel([0.597975, -1.435098, -2.536750, -0.740541, 1.570796, 2.168772],accel_mss,speed_ms,0,blend_radius_m)
    |   movel([0.600763, -1.433280, -2.538175, -0.740934, 1.570796, 2.171559],accel_mss,speed_ms,0,blend_radius_m)
    |   movel([0.603602, -1.431531, -2.539540, -0.741318, 1.570796, 2.174399],accel_mss,speed_ms,0,blend_radius_m)
    |   movel([0.609428, -1.428210, -2.542121, -0.742058, 1.570796, 2.180224],accel_mss,speed_ms,0,blend_radius_m)
    |   movel([0.607327, -1.428865, -2.541613, -0.741911, 1.570796, 2.178123],accel_mss,speed_ms,0,blend_radius_m)
    |   movel([0.601055, -1.430361, -2.540452, -0.741577, 1.570796, 2.171851],accel_mss,speed_ms,0,blend_radius_m)
    |   movel([0.598948, -1.430939, -2.540001, -0.741448, 1.570796, 2.169745],accel_mss,speed_ms,0,blend_radius_m)
    |   movel([0.596838, -1.431670, -2.539432, -0.741287, 1.570796, 2.167634],accel_mss,speed_ms,0,blend_radius_m)
    |   movel([0.594769, -1.432599, -2.538707, -0.741083, 1.570796, 2.165565],accel_mss,speed_ms,0,blend_radius_m)
    |   movel([0.592779, -1.433776, -2.537787, -0.740827, 1.570796, 2.163576],accel_mss,speed_ms,0,blend_radius_m)
    |   movel([0.595779, -1.431504, -2.539561, -0.741324, 1.570796, 2.166575],accel_mss,speed_ms,0,blend_radius_m)
    |   movel([0.598829, -1.429078, -2.541448, -0.741863, 1.570796, 2.169625],accel_mss,speed_ms,0,blend_radius_m)
    |   movel([0.601939, -1.426743, -2.543256, -0.742390, 1.570796, 2.172735],accel_mss,speed_ms,0,blend_radius_m)
    |   movel([0.603516, -1.425689, -2.544069, -0.742631, 1.570796, 2.174312],accel_mss,speed_ms,0,blend_radius_m)
    |   movel([0.605110, -1.424755, -2.544788, -0.742846, 1.570796, 2.175906],accel_mss,speed_ms,0,blend_radius_m)
    |   movel([0.610674, -1.421976, -2.546920, -0.743493, 1.570796, 2.181470],accel_mss,speed_ms,0,blend_radius_m)
    |   movel([0.616281, -1.419292, -2.548968, -0.744129, 1.570796, 2.187077],accel_mss,speed_ms,0,blend_radius_m)
    |   movel([0.612807, -1.419908, -2.548499, -0.743982, 1.570796, 2.183604],accel_mss,speed_ms,0,blend_radius_m)
    |   movel([0.609513, -1.420785, -2.547830, -0.743774, 1.570796, 2.180309],accel_mss,speed_ms,0,blend_radius_m)
    |   movel([0.606185, -1.421997, -2.546904, -0.743488, 1.570796, 2.176982],accel_mss,speed_ms,0,blend_radius_m)
    |   movel([0.602617, -1.423612, -2.545666, -0.743111, 1.570796, 2.173414],accel_mss,speed_ms,0,blend_radius_m)
    |   movel([0.604426, -1.422617, -2.546429, -0.743343, 1.570796, 2.175222],accel_mss,speed_ms,0,blend_radius_m)
    |   movel([0.606160, -1.421478, -2.547301, -0.743610, 1.570796, 2.176957],accel_mss,speed_ms,0,blend_radius_m)
    |   movel([0.612874, -1.416370, -2.551186, -0.744833, 1.570796, 2.183671],accel_mss,speed_ms,0,blend_radius_m)
    |   movel([0.614624, -1.415179, -2.552086, -0.745124, 1.570796, 2.185420],accel_mss,speed_ms,0,blend_radius_m)
    |   movel([0.616455, -1.414116, -2.552888, -0.745386, 1.570796, 2.187252],accel_mss,speed_ms,0,blend_radius_m)
    |   movel([0.618929, -1.412961, -2.553757, -0.745671, 1.570796, 2.189725],accel_mss,speed_ms,0,blend_radius_m)
    |   movel([0.620899, -1.412360, -2.554208, -0.745821, 1.570796, 2.191696],accel_mss,speed_ms,0,blend_radius_m)
    |   movel([0.621394, -1.412105, -2.554399, -0.745885, 1.570796, 2.192190],accel_mss,speed_ms,0,blend_radius_m)
    |   movel([0.621694, -1.411717, -2.554690, -0.745981, 1.570796, 2.192491],accel_mss,speed_ms,0,blend_radius_m)
    |   movel([0.621604, -1.411410, -2.554921, -0.746058, 1.570796, 2.192400],accel_mss,speed_ms,0,blend_radius_m)
    |   movel([0.621218, -1.411175, -2.555097, -0.746117, 1.570796, 2.192015],accel_mss,speed_ms,0,blend_radius_m)
    |   movel([0.620633, -1.411008, -2.555222, -0.746159, 1.570796, 2.191429],accel_mss,speed_ms,0,blend_radius_m)
    |   movel([0.619253, -1.410833, -2.555353, -0.746203, 1.570796, 2.190050],accel_mss,speed_ms,0,blend_radius_m)
    |   movel([0.618236, -1.410821, -2.555361, -0.746206, 1.570796, 2.189032],accel_mss,speed_ms,0,blend_radius_m)
    |   movel([0.620369, -1.409639, -2.556245, -0.746505, 1.570796, 2.191165],accel_mss,speed_ms,0,blend_radius_m)
    |   movel([0.622664, -1.408686, -2.556956, -0.746747, 1.570796, 2.193460],accel_mss,speed_ms,0,blend_radius_m)
    |   movel([0.627198, -1.407232, -2.558038, -0.747119, 1.570796, 2.197994],accel_mss,speed_ms,0,blend_radius_m)
    |   speed_ms = 0.005
    |   movel([0.627198, -1.398614, -2.554165, -0.759610, 1.570796, 2.197994],accel_mss,speed_ms,0,blend_radius_m)
    |   speed_ms = 0.040
    |   movel([0.620757, -1.396853, -2.555454, -0.760082, 1.570796, 2.191554],accel_mss,speed_ms,0,blend_radius_m)
    |   speed_ms = 0.005
    |   movel([0.620757, -1.405485, -2.559334, -0.747570, 1.570796, 2.191554],accel_mss,speed_ms,0,blend_radius_m)
    |   speed_ms = 0.025
    |   movel([0.620686, -1.404286, -2.560221, -0.747882, 1.570796, 2.191483],accel_mss,speed_ms,0,blend_radius_m)
    |   movel([0.620351, -1.403242, -2.560991, -0.748156, 1.570796, 2.191147],accel_mss,speed_ms,0,blend_radius_m)
    |   movel([0.619786, -1.402345, -2.561651, -0.748392, 1.570796, 2.190582],accel_mss,speed_ms,0,blend_radius_m)
    |   movel([0.619029, -1.401586, -2.562210, -0.748593, 1.570796, 2.189825],accel_mss,speed_ms,0,blend_radius_m)
    |   movel([0.618111, -1.400959, -2.562670, -0.748760, 1.570796, 2.188907],accel_mss,speed_ms,0,blend_radius_m)
    |   movel([0.617070, -1.400457, -2.563038, -0.748894, 1.570796, 2.187866],accel_mss,speed_ms,0,blend_radius_m)
    |   movel([0.614756, -1.399786, -2.563530, -0.749073, 1.570796, 2.185552],accel_mss,speed_ms,0,blend_radius_m)
    |   speed_ms = 0.005
    |   movel([0.614756, -1.391112, -2.559625, -0.761652, 1.570796, 2.185552],accel_mss,speed_ms,0,blend_radius_m)
    |   speed_ms = 0.040
    |   movel([0.625725, -1.390491, -2.560073, -0.761825, 1.570796, 2.196521],accel_mss,speed_ms,0,blend_radius_m)
    |   speed_ms = 0.005
    |   movel([0.625725, -1.399170, -2.563981, -0.749239, 1.570796, 2.196521],accel_mss,speed_ms,0,blend_radius_m)
    |   speed_ms = 0.025
    |   movel([0.626265, -1.397103, -2.565489, -0.749798, 1.570796, 2.197062],accel_mss,speed_ms,0,blend_radius_m)
    |   movel([0.626659, -1.395120, -2.566930, -0.750340, 1.570796, 2.197455],accel_mss,speed_ms,0,blend_radius_m)
    |   movel([0.626847, -1.393251, -2.568282, -0.750856, 1.570796, 2.197643],accel_mss,speed_ms,0,blend_radius_m)
    |   movel([0.626773, -1.391522, -2.569529, -0.751338, 1.570796, 2.197569],accel_mss,speed_ms,0,blend_radius_m)
    |   movel([0.626372, -1.389972, -2.570643, -0.751774, 1.570796, 2.197168],accel_mss,speed_ms,0,blend_radius_m)
    |   movel([0.625594, -1.388623, -2.571610, -0.752156, 1.570796, 2.196390],accel_mss,speed_ms,0,blend_radius_m)
    |   movel([0.624373, -1.387515, -2.572402, -0.752472, 1.570796, 2.195169],accel_mss,speed_ms,0,blend_radius_m)
    |   movel([0.623579, -1.387059, -2.572728, -0.752602, 1.570796, 2.194376],accel_mss,speed_ms,0,blend_radius_m)
    |   movel([0.622653, -1.386675, -2.573001, -0.752712, 1.570796, 2.193449],accel_mss,speed_ms,0,blend_radius_m)
    |   speed_ms = 0.005
    |   movel([0.622653, -1.377905, -2.569039, -0.765445, 1.570796, 2.193449],accel_mss,speed_ms,0,blend_radius_m)
    |   speed_ms = 0.040
    |   movel([0.631539, -1.377852, -2.569076, -0.765461, 1.570796, 2.202335],accel_mss,speed_ms,0,blend_radius_m)
    |   speed_ms = 0.005
    |   movel([0.631539, -1.386623, -2.573039, -0.752727, 1.570796, 2.202335],accel_mss,speed_ms,0,blend_radius_m)
    |   speed_ms = 0.025
    |   movel([0.633312, -1.382368, -2.576058, -0.753963, 1.570796, 2.204109],accel_mss,speed_ms,0,blend_radius_m)
    |   movel([0.633980, -1.380300, -2.577517, -0.754573, 1.570796, 2.204776],accel_mss,speed_ms,0,blend_radius_m)
    |   movel([0.634421, -1.378299, -2.578922, -0.755169, 1.570796, 2.205218],accel_mss,speed_ms,0,blend_radius_m)
    |   movel([0.634579, -1.376391, -2.580255, -0.755742, 1.570796, 2.205375],accel_mss,speed_ms,0,blend_radius_m)
    |   movel([0.634391, -1.374604, -2.581500, -0.756284, 1.570796, 2.205187],accel_mss,speed_ms,0,blend_radius_m)
    |   movel([0.633797, -1.372957, -2.582644, -0.756788, 1.570796, 2.204594],accel_mss,speed_ms,0,blend_radius_m)
    |   movel([0.632737, -1.371480, -2.583666, -0.757243, 1.570796, 2.203533],accel_mss,speed_ms,0,blend_radius_m)
    |   speed_ms = 0.005
    |   movel([0.632737, -1.362601, -2.579637, -0.770152, 1.570796, 2.203533],accel_mss,speed_ms,0,blend_radius_m)
    |   speed_ms = 0.040
    |   movel([0.638756, -1.366287, -2.577114, -0.768988, 1.570796, 2.209552],accel_mss,speed_ms,0,blend_radius_m)
    |   speed_ms = 0.005
    |   movel([0.638756, -1.375140, -2.581128, -0.756121, 1.570796, 2.209552],accel_mss,speed_ms,0,blend_radius_m)
    |   speed_ms = 0.025
    |   movel([0.640325, -1.372678, -2.582837, -0.756873, 1.570796, 2.211122],accel_mss,speed_ms,0,blend_radius_m)
    |   movel([0.641788, -1.370130, -2.584598, -0.757661, 1.570796, 2.212584],accel_mss,speed_ms,0,blend_radius_m)
    |   movel([0.643066, -1.367539, -2.586378, -0.758472, 1.570796, 2.213862],accel_mss,speed_ms,0,blend_radius_m)
    |   movel([0.644082, -1.364961, -2.588140, -0.759288, 1.570796, 2.214878],accel_mss,speed_ms,0,blend_radius_m)
    |   movel([0.644761, -1.362438, -2.589855, -0.760095, 1.570796, 2.215558],accel_mss,speed_ms,0,blend_radius_m)
    |   movel([0.644947, -1.361216, -2.590683, -0.760490, 1.570796, 2.215744],accel_mss,speed_ms,0,blend_radius_m)
    |   movel([0.644972, -1.358881, -2.592258, -0.761249, 1.570796, 2.215768],accel_mss,speed_ms,0,blend_radius_m)
    |   movel([0.644788, -1.357782, -2.592997, -0.761610, 1.570796, 2.215584],accel_mss,speed_ms,0,blend_radius_m)
    |   movel([0.644460, -1.356735, -2.593700, -0.761954, 1.570796, 2.215256],accel_mss,speed_ms,0,blend_radius_m)
    |   movel([0.643978, -1.355752, -2.594358, -0.762279, 1.570796, 2.214774],accel_mss,speed_ms,0,blend_radius_m)
    |   speed_ms = 0.005
    |   movel([0.643978, -1.346763, -2.590258, -0.775368, 1.570796, 2.214774],accel_mss,speed_ms,0,blend_radius_m)
    |   speed_ms = 0.040
    |   movel([0.650408, -1.350380, -2.587863, -0.774146, 1.570796, 2.221204],accel_mss,speed_ms,0,blend_radius_m)
    |   speed_ms = 0.005
    |   movel([0.650408, -1.359345, -2.591946, -0.761098, 1.570796, 2.221204],accel_mss,speed_ms,0,blend_radius_m)
    |   speed_ms = 0.025
    |   movel([0.652391, -1.356509, -2.593851, -0.762029, 1.570796, 2.223187],accel_mss,speed_ms,0,blend_radius_m)
    |   movel([0.654173, -1.353565, -2.595817, -0.763007, 1.570796, 2.224970],accel_mss,speed_ms,0,blend_radius_m)
    |   movel([0.655681, -1.350573, -2.597802, -0.764014, 1.570796, 2.226477],accel_mss,speed_ms,0,blend_radius_m)
    |   movel([0.656825, -1.347599, -2.599763, -0.765027, 1.570796, 2.227621],accel_mss,speed_ms,0,blend_radius_m)
    |   movel([0.657528, -1.344707, -2.601658, -0.766024, 1.570796, 2.228325],accel_mss,speed_ms,0,blend_radius_m)
    |   movel([0.657685, -1.343314, -2.602567, -0.766508, 1.570796, 2.228481],accel_mss,speed_ms,0,blend_radius_m)
    |   movel([0.657703, -1.341966, -2.603444, -0.766979, 1.570796, 2.228499],accel_mss,speed_ms,0,blend_radius_m)
    |   movel([0.657564, -1.340675, -2.604281, -0.767433, 1.570796, 2.228360],accel_mss,speed_ms,0,blend_radius_m)
    |   movel([0.657263, -1.339444, -2.605078, -0.767868, 1.570796, 2.228060],accel_mss,speed_ms,0,blend_radius_m)
    |   movel([0.656787, -1.338289, -2.605822, -0.768277, 1.570796, 2.227583],accel_mss,speed_ms,0,blend_radius_m)
    |   movel([0.656126, -1.337213, -2.606515, -0.768661, 1.570796, 2.226923],accel_mss,speed_ms,0,blend_radius_m)
    |   speed_ms = 0.005
    |   movel([0.656126, -1.328100, -2.602333, -0.781957, 1.570796, 2.226923],accel_mss,speed_ms,0,blend_radius_m)
    |   speed_ms = 0.040
    |   movel([0.621666, -1.319357, -2.607827, -0.785205, 1.570796, 2.192462],accel_mss,speed_ms,0,blend_radius_m)
    |   speed_ms = 0.005
    |   movel([0.621666, -1.328527, -2.612049, -0.771813, 1.570796, 2.192462],accel_mss,speed_ms,0,blend_radius_m)
    |   speed_ms = 0.025
    |   movel([0.622565, -1.330597, -2.610739, -0.771053, 1.570796, 2.193361],accel_mss,speed_ms,0,blend_radius_m)
    |   movel([0.623171, -1.332843, -2.609312, -0.770234, 1.570796, 2.193967],accel_mss,speed_ms,0,blend_radius_m)
    |   movel([0.623505, -1.335243, -2.607779, -0.769367, 1.570796, 2.194301],accel_mss,speed_ms,0,blend_radius_m)
    |   movel([0.623585, -1.337774, -2.606154, -0.768461, 1.570796, 2.194382],accel_mss,speed_ms,0,blend_radius_m)
    |   movel([0.623426, -1.340411, -2.604452, -0.767526, 1.570796, 2.194222],accel_mss,speed_ms,0,blend_radius_m)
    |   movel([0.623051, -1.343134, -2.602684, -0.766571, 1.570796, 2.193847],accel_mss,speed_ms,0,blend_radius_m)
    |   movel([0.622469, -1.345924, -2.600862, -0.765603, 1.570796, 2.193266],accel_mss,speed_ms,0,blend_radius_m)
    |   movel([0.621708, -1.348755, -2.599002, -0.764632, 1.570796, 2.192504],accel_mss,speed_ms,0,blend_radius_m)
    |   movel([0.620776, -1.351608, -2.597117, -0.763664, 1.570796, 2.191572],accel_mss,speed_ms,0,blend_radius_m)
    |   movel([0.619696, -1.354465, -2.595217, -0.762707, 1.570796, 2.190492],accel_mss,speed_ms,0,blend_radius_m)
    |   movel([0.618481, -1.357303, -2.593319, -0.761767, 1.570796, 2.189278],accel_mss,speed_ms,0,blend_radius_m)
    |   movel([0.617148, -1.360107, -2.591432, -0.760850, 1.570796, 2.187944],accel_mss,speed_ms,0,blend_radius_m)
    |   movel([0.615715, -1.362853, -2.589574, -0.759962, 1.570796, 2.186512],accel_mss,speed_ms,0,blend_radius_m)
    |   movel([0.614192, -1.365529, -2.587753, -0.759107, 1.570796, 2.184989],accel_mss,speed_ms,0,blend_radius_m)
    |   movel([0.612601, -1.368109, -2.585988, -0.758293, 1.570796, 2.183397],accel_mss,speed_ms,0,blend_radius_m)
    |   movel([0.610954, -1.370581, -2.584286, -0.757521, 1.570796, 2.181750],accel_mss,speed_ms,0,blend_radius_m)
    |   movel([0.608645, -1.373803, -2.582057, -0.756529, 1.570796, 2.179441],accel_mss,speed_ms,0,blend_radius_m)
    |   movel([0.605844, -1.377409, -2.579544, -0.755436, 1.570796, 2.176640],accel_mss,speed_ms,0,blend_radius_m)
    |   movel([0.602687, -1.381032, -2.577001, -0.754356, 1.570796, 2.173483],accel_mss,speed_ms,0,blend_radius_m)
    |   movel([0.601016, -1.382739, -2.575796, -0.753854, 1.570796, 2.171812],accel_mss,speed_ms,0,blend_radius_m)
    |   movel([0.599309, -1.384316, -2.574679, -0.753394, 1.570796, 2.170106],accel_mss,speed_ms,0,blend_radius_m)
    |   movel([0.597574, -1.385721, -2.573681, -0.752987, 1.570796, 2.168370],accel_mss,speed_ms,0,blend_radius_m)
    |   movel([0.595833, -1.386908, -2.572835, -0.752646, 1.570796, 2.166630],accel_mss,speed_ms,0,blend_radius_m)
    |   movel([0.594095, -1.387836, -2.572173, -0.752380, 1.570796, 2.164892],accel_mss,speed_ms,0,blend_radius_m)
    |   movel([0.592375, -1.388464, -2.571724, -0.752201, 1.570796, 2.163171],accel_mss,speed_ms,0,blend_radius_m)
    |   movel([0.590691, -1.388744, -2.571523, -0.752121, 1.570796, 2.161487],accel_mss,speed_ms,0,blend_radius_m)
    |   movel([0.589052, -1.388638, -2.571599, -0.752152, 1.570796, 2.159848],accel_mss,speed_ms,0,blend_radius_m)
    |   movel([0.588253, -1.388424, -2.571753, -0.752213, 1.570796, 2.159050],accel_mss,speed_ms,0,blend_radius_m)
    |   movel([0.587471, -1.388096, -2.571987, -0.752306, 1.570796, 2.158268],accel_mss,speed_ms,0,blend_radius_m)
    |   movel([0.585965, -1.387077, -2.572715, -0.752597, 1.570796, 2.156761],accel_mss,speed_ms,0,blend_radius_m)
    |   movel([0.584424, -1.385537, -2.573812, -0.753040, 1.570796, 2.155220],accel_mss,speed_ms,0,blend_radius_m)
    |   movel([0.583153, -1.383849, -2.575010, -0.753530, 1.570796, 2.153949],accel_mss,speed_ms,0,blend_radius_m)
    |   movel([0.582122, -1.382027, -2.576299, -0.754063, 1.570796, 2.152918],accel_mss,speed_ms,0,blend_radius_m)
    |   movel([0.581300, -1.380074, -2.577675, -0.754640, 1.570796, 2.152096],accel_mss,speed_ms,0,blend_radius_m)
    |   movel([0.580659, -1.378000, -2.579131, -0.755258, 1.570796, 2.151455],accel_mss,speed_ms,0,blend_radius_m)
    |   movel([0.580165, -1.375815, -2.580658, -0.755917, 1.570796, 2.150961],accel_mss,speed_ms,0,blend_radius_m)
    |   movel([0.579497, -1.371134, -2.583905, -0.757350, 1.570796, 2.150294],accel_mss,speed_ms,0,blend_radius_m)
    |   movel([0.578951, -1.365850, -2.587534, -0.759005, 1.570796, 2.149747],accel_mss,speed_ms,0,blend_radius_m)
    |   movel([0.578551, -1.360508, -2.591161, -0.760719, 1.570796, 2.149347],accel_mss,speed_ms,0,blend_radius_m)
    |   movel([0.578456, -1.355007, -2.594855, -0.762526, 1.570796, 2.149252],accel_mss,speed_ms,0,blend_radius_m)
    |   movel([0.578578, -1.352162, -2.596749, -0.763478, 1.570796, 2.149375],accel_mss,speed_ms,0,blend_radius_m)
    |   movel([0.578843, -1.349233, -2.598687, -0.764469, 1.570796, 2.149640],accel_mss,speed_ms,0,blend_radius_m)
    |   movel([0.579128, -1.345588, -2.601082, -0.765719, 1.570796, 2.149924],accel_mss,speed_ms,0,blend_radius_m)
    |   movel([0.579166, -1.341949, -2.603455, -0.766985, 1.570796, 2.149962],accel_mss,speed_ms,0,blend_radius_m)
    |   movel([0.578983, -1.338332, -2.605795, -0.768262, 1.570796, 2.149780],accel_mss,speed_ms,0,blend_radius_m)
    |   movel([0.578620, -1.334746, -2.608097, -0.769545, 1.570796, 2.149417],accel_mss,speed_ms,0,blend_radius_m)
    |   movel([0.577474, -1.327732, -2.612550, -0.772107, 1.570796, 2.148271],accel_mss,speed_ms,0,blend_radius_m)
    |   movel([0.576003, -1.321005, -2.616758, -0.774626, 1.570796, 2.146800],accel_mss,speed_ms,0,blend_radius_m)
    |   movel([0.574612, -1.316084, -2.619798, -0.776507, 1.570796, 2.145408],accel_mss,speed_ms,0,blend_radius_m)
    |   movel([0.572792, -1.311386, -2.622670, -0.778332, 1.570796, 2.143588],accel_mss,speed_ms,0,blend_radius_m)
    |   movel([0.570532, -1.306949, -2.625357, -0.780084, 1.570796, 2.141328],accel_mss,speed_ms,0,blend_radius_m)
    |   movel([0.567821, -1.302820, -2.627833, -0.781736, 1.570796, 2.138617],accel_mss,speed_ms,0,blend_radius_m)
    |   movel([0.564652, -1.299032, -2.630085, -0.783272, 1.570796, 2.135448],accel_mss,speed_ms,0,blend_radius_m)
    |   movel([0.562893, -1.297282, -2.631119, -0.783988, 1.570796, 2.133689],accel_mss,speed_ms,0,blend_radius_m)
    |   movel([0.559022, -1.294091, -2.632994, -0.785303, 1.570796, 2.129818],accel_mss,speed_ms,0,blend_radius_m)
    |   movel([0.556907, -1.292661, -2.633831, -0.785897, 1.570796, 2.127704],accel_mss,speed_ms,0,blend_radius_m)
    |   movel([0.552322, -1.290161, -2.635286, -0.786941, 1.570796, 2.123118],accel_mss,speed_ms,0,blend_radius_m)
    |   movel([0.548890, -1.288814, -2.636068, -0.787508, 1.570796, 2.119686],accel_mss,speed_ms,0,blend_radius_m)
    |   movel([0.545173, -1.287852, -2.636624, -0.787913, 1.570796, 2.115969],accel_mss,speed_ms,0,blend_radius_m)
    |   movel([0.541202, -1.287290, -2.636948, -0.788150, 1.570796, 2.111998],accel_mss,speed_ms,0,blend_radius_m)
    |   movel([0.537005, -1.287149, -2.637030, -0.788210, 1.570796, 2.107801],accel_mss,speed_ms,0,blend_radius_m)
    |   movel([0.532609, -1.287443, -2.636860, -0.788086, 1.570796, 2.103406],accel_mss,speed_ms,0,blend_radius_m)
    |   movel([0.528049, -1.288183, -2.636433, -0.787773, 1.570796, 2.098845],accel_mss,speed_ms,0,blend_radius_m)
    |   movel([0.523356, -1.289383, -2.635738, -0.787268, 1.570796, 2.094152],accel_mss,speed_ms,0,blend_radius_m)
    |   movel([0.518564, -1.291050, -2.634770, -0.786569, 1.570796, 2.089360],accel_mss,speed_ms,0,blend_radius_m)
    |   movel([0.514066, -1.292974, -2.633648, -0.785767, 1.570796, 2.084862],accel_mss,speed_ms,0,blend_radius_m)
    |   movel([0.509727, -1.295149, -2.632374, -0.784866, 1.570796, 2.080523],accel_mss,speed_ms,0,blend_radius_m)
    |   movel([0.505563, -1.297588, -2.630938, -0.783862, 1.570796, 2.076360],accel_mss,speed_ms,0,blend_radius_m)
    |   movel([0.501589, -1.300304, -2.629331, -0.782754, 1.570796, 2.072386],accel_mss,speed_ms,0,blend_radius_m)
    |   movel([0.499677, -1.301770, -2.628459, -0.782160, 1.570796, 2.070473],accel_mss,speed_ms,0,blend_radius_m)
    |   movel([0.496018, -1.304922, -2.626575, -0.780892, 1.570796, 2.066815],accel_mss,speed_ms,0,blend_radius_m)
    |   movel([0.494274, -1.306613, -2.625559, -0.780217, 1.570796, 2.065071],accel_mss,speed_ms,0,blend_radius_m)
    |   movel([0.490969, -1.310226, -2.623376, -0.778788, 1.570796, 2.061765],accel_mss,speed_ms,0,blend_radius_m)
    |   movel([0.489409, -1.312153, -2.622204, -0.778032, 1.570796, 2.060205],accel_mss,speed_ms,0,blend_radius_m)
    |   movel([0.487917, -1.314158, -2.620980, -0.777252, 1.570796, 2.058713],accel_mss,speed_ms,0,blend_radius_m)
    |   movel([0.485915, -1.317093, -2.619178, -0.776118, 1.570796, 2.056711],accel_mss,speed_ms,0,blend_radius_m)
    |   movel([0.484053, -1.320085, -2.617329, -0.774975, 1.570796, 2.054849],accel_mss,speed_ms,0,blend_radius_m)
    |   movel([0.482333, -1.323108, -2.615449, -0.773832, 1.570796, 2.053129],accel_mss,speed_ms,0,blend_radius_m)
    |   movel([0.480751, -1.326147, -2.613547, -0.772695, 1.570796, 2.051547],accel_mss,speed_ms,0,blend_radius_m)
    |   movel([0.479315, -1.329177, -2.611638, -0.771574, 1.570796, 2.050111],accel_mss,speed_ms,0,blend_radius_m)
    |   movel([0.478026, -1.332177, -2.609736, -0.770476, 1.570796, 2.048823],accel_mss,speed_ms,0,blend_radius_m)
    |   movel([0.476884, -1.335130, -2.607852, -0.769407, 1.570796, 2.047680],accel_mss,speed_ms,0,blend_radius_m)
    |   movel([0.475891, -1.338015, -2.605999, -0.768375, 1.570796, 2.046688],accel_mss,speed_ms,0,blend_radius_m)
    |   movel([0.472966, -1.349149, -2.598742, -0.764497, 1.570796, 2.043762],accel_mss,speed_ms,0,blend_radius_m)
    |   movel([0.470619, -1.357979, -2.592865, -0.761545, 1.570796, 2.041416],accel_mss,speed_ms,0,blend_radius_m)
    |   movel([0.470325, -1.358818, -2.592301, -0.761270, 1.570796, 2.041122],accel_mss,speed_ms,0,blend_radius_m)
    |   movel([0.475631, -1.356833, -2.593634, -0.761922, 1.570796, 2.046427],accel_mss,speed_ms,0,blend_radius_m)
    |   movel([0.480943, -1.355196, -2.594729, -0.762464, 1.570796, 2.051739],accel_mss,speed_ms,0,blend_radius_m)
    |   movel([0.486236, -1.353899, -2.595594, -0.762896, 1.570796, 2.057033],accel_mss,speed_ms,0,blend_radius_m)
    |   movel([0.491479, -1.352929, -2.596240, -0.763220, 1.570796, 2.062275],accel_mss,speed_ms,0,blend_radius_m)
    |   movel([0.496639, -1.352279, -2.596672, -0.763438, 1.570796, 2.067435],accel_mss,speed_ms,0,blend_radius_m)
    |   movel([0.501690, -1.351932, -2.596902, -0.763555, 1.570796, 2.072486],accel_mss,speed_ms,0,blend_radius_m)
    |   movel([0.506601, -1.351881, -2.596936, -0.763573, 1.570796, 2.077398],accel_mss,speed_ms,0,blend_radius_m)
    |   movel([0.511345, -1.352106, -2.596786, -0.763497, 1.570796, 2.082141],accel_mss,speed_ms,0,blend_radius_m)
    |   movel([0.513503, -1.352345, -2.596628, -0.763416, 1.570796, 2.084300],accel_mss,speed_ms,0,blend_radius_m)
    |   movel([0.515622, -1.352729, -2.596373, -0.763287, 1.570796, 2.086418],accel_mss,speed_ms,0,blend_radius_m)
    |   movel([0.517679, -1.353257, -2.596022, -0.763110, 1.570796, 2.088475],accel_mss,speed_ms,0,blend_radius_m)
    |   movel([0.519651, -1.353929, -2.595574, -0.762885, 1.570796, 2.090447],accel_mss,speed_ms,0,blend_radius_m)
    |   movel([0.521517, -1.354747, -2.595029, -0.762613, 1.570796, 2.092314],accel_mss,speed_ms,0,blend_radius_m)
    |   movel([0.523257, -1.355711, -2.594385, -0.762293, 1.570796, 2.094053],accel_mss,speed_ms,0,blend_radius_m)
    |   movel([0.524849, -1.356818, -2.593644, -0.761927, 1.570796, 2.095645],accel_mss,speed_ms,0,blend_radius_m)
    |   movel([0.526273, -1.358067, -2.592806, -0.761516, 1.570796, 2.097069],accel_mss,speed_ms,0,blend_radius_m)
    |   movel([0.527508, -1.359460, -2.591868, -0.761060, 1.570796, 2.098304],accel_mss,speed_ms,0,blend_radius_m)
    |   movel([0.528536, -1.360996, -2.590832, -0.760561, 1.570796, 2.099332],accel_mss,speed_ms,0,blend_radius_m)
    |   movel([0.529334, -1.362671, -2.589697, -0.760020, 1.570796, 2.100130],accel_mss,speed_ms,0,blend_radius_m)
    |   movel([0.529883, -1.364486, -2.588464, -0.759439, 1.570796, 2.100680],accel_mss,speed_ms,0,blend_radius_m)
    |   movel([0.530165, -1.366437, -2.587133, -0.758820, 1.570796, 2.100962],accel_mss,speed_ms,0,blend_radius_m)
    |   movel([0.530163, -1.368526, -2.585701, -0.758162, 1.570796, 2.100960],accel_mss,speed_ms,0,blend_radius_m)
    |   movel([0.529857, -1.370747, -2.584172, -0.757470, 1.570796, 2.100654],accel_mss,speed_ms,0,blend_radius_m)
    |   movel([0.529228, -1.373102, -2.582544, -0.756743, 1.570796, 2.100024],accel_mss,speed_ms,0,blend_radius_m)
    |   movel([0.528005, -1.376258, -2.580348, -0.755782, 1.570796, 2.098801],accel_mss,speed_ms,0,blend_radius_m)
    |   movel([0.526428, -1.379471, -2.578099, -0.754819, 1.570796, 2.097224],accel_mss,speed_ms,0,blend_radius_m)
    |   movel([0.524564, -1.382702, -2.575822, -0.753865, 1.570796, 2.095360],accel_mss,speed_ms,0,blend_radius_m)
    |   movel([0.522477, -1.385922, -2.573537, -0.752929, 1.570796, 2.093273],accel_mss,speed_ms,0,blend_radius_m)
    |   movel([0.520232, -1.389098, -2.571270, -0.752021, 1.570796, 2.091028],accel_mss,speed_ms,0,blend_radius_m)
    |   movel([0.517887, -1.392198, -2.569042, -0.751149, 1.570796, 2.088683],accel_mss,speed_ms,0,blend_radius_m)
    |   movel([0.513159, -1.398048, -2.564800, -0.749541, 1.570796, 2.083955],accel_mss,speed_ms,0,blend_radius_m)
    |   movel([0.510054, -1.401623, -2.562183, -0.748583, 1.570796, 2.080850],accel_mss,speed_ms,0,blend_radius_m)
    |   movel([0.506857, -1.405036, -2.559666, -0.747687, 1.570796, 2.077653],accel_mss,speed_ms,0,blend_radius_m)
    |   movel([0.503577, -1.408310, -2.557236, -0.746843, 1.570796, 2.074373],accel_mss,speed_ms,0,blend_radius_m)
    |   movel([0.500217, -1.411476, -2.554871, -0.746042, 1.570796, 2.071013],accel_mss,speed_ms,0,blend_radius_m)
    |   movel([0.496786, -1.414553, -2.552558, -0.745278, 1.570796, 2.067583],accel_mss,speed_ms,0,blend_radius_m)
    |   movel([0.493292, -1.417568, -2.550278, -0.744543, 1.570796, 2.064088],accel_mss,speed_ms,0,blend_radius_m)
    |   movel([0.486129, -1.423508, -2.545746, -0.743135, 1.570796, 2.056925],accel_mss,speed_ms,0,blend_radius_m)
    |   movel([0.487951, -1.426525, -2.543424, -0.742440, 1.570796, 2.058747],accel_mss,speed_ms,0,blend_radius_m)
    |   movel([0.488812, -1.428211, -2.542120, -0.742058, 1.570796, 2.059609],accel_mss,speed_ms,0,blend_radius_m)
    |   movel([0.489370, -1.429952, -2.540769, -0.741667, 1.570796, 2.060166],accel_mss,speed_ms,0,blend_radius_m)
    |   movel([0.489470, -1.430830, -2.540087, -0.741472, 1.570796, 2.060266],accel_mss,speed_ms,0,blend_radius_m)
    |   movel([0.489417, -1.431705, -2.539405, -0.741279, 1.570796, 2.060213],accel_mss,speed_ms,0,blend_radius_m)
    |   movel([0.489187, -1.432571, -2.538729, -0.741089, 1.570796, 2.059983],accel_mss,speed_ms,0,blend_radius_m)
    |   movel([0.488755, -1.433422, -2.538064, -0.740904, 1.570796, 2.059551],accel_mss,speed_ms,0,blend_radius_m)
    |   movel([0.488098, -1.434250, -2.537415, -0.740724, 1.570796, 2.058895],accel_mss,speed_ms,0,blend_radius_m)
    |   movel([0.487186, -1.435055, -2.536784, -0.740550, 1.570796, 2.057983],accel_mss,speed_ms,0,blend_radius_m)
    |   movel([0.485997, -1.435830, -2.536175, -0.740384, 1.570796, 2.056793],accel_mss,speed_ms,0,blend_radius_m)
    |   movel([0.484506, -1.436568, -2.535594, -0.740227, 1.570796, 2.055302],accel_mss,speed_ms,0,blend_radius_m)
    |   movel([0.483220, -1.437075, -2.535195, -0.740119, 1.570796, 2.054016],accel_mss,speed_ms,0,blend_radius_m)
    |   movel([0.482001, -1.437448, -2.534901, -0.740040, 1.570796, 2.052798],accel_mss,speed_ms,0,blend_radius_m)
    |   movel([0.480845, -1.437700, -2.534702, -0.739987, 1.570796, 2.051642],accel_mss,speed_ms,0,blend_radius_m)
    |   movel([0.478697, -1.437878, -2.534562, -0.739949, 1.570796, 2.049493],accel_mss,speed_ms,0,blend_radius_m)
    |   movel([0.477695, -1.437824, -2.534604, -0.739961, 1.570796, 2.048491],accel_mss,speed_ms,0,blend_radius_m)
    |   movel([0.475806, -1.437485, -2.534871, -0.740032, 1.570796, 2.046602],accel_mss,speed_ms,0,blend_radius_m)
    |   movel([0.474040, -1.436905, -2.535329, -0.740155, 1.570796, 2.044837],accel_mss,speed_ms,0,blend_radius_m)
    |   movel([0.472356, -1.436162, -2.535914, -0.740313, 1.570796, 2.043153],accel_mss,speed_ms,0,blend_radius_m)
    |   movel([0.469076, -1.434521, -2.537203, -0.740665, 1.570796, 2.039872],accel_mss,speed_ms,0,blend_radius_m)
    |   movel([0.465722, -1.436483, -2.535661, -0.740245, 1.570796, 2.036518],accel_mss,speed_ms,0,blend_radius_m)
    |   movel([0.463980, -1.437385, -2.534950, -0.740053, 1.570796, 2.034776],accel_mss,speed_ms,0,blend_radius_m)
    |   movel([0.462220, -1.438181, -2.534322, -0.739885, 1.570796, 2.033016],accel_mss,speed_ms,0,blend_radius_m)
    |   movel([0.460464, -1.438828, -2.533812, -0.739750, 1.570796, 2.031260],accel_mss,speed_ms,0,blend_radius_m)
    |   movel([0.458733, -1.439284, -2.533451, -0.739654, 1.570796, 2.029530],accel_mss,speed_ms,0,blend_radius_m)
    |   movel([0.457049, -1.439507, -2.533274, -0.739608, 1.570796, 2.027846],accel_mss,speed_ms,0,blend_radius_m)
    |   movel([0.455428, -1.439456, -2.533315, -0.739619, 1.570796, 2.026225],accel_mss,speed_ms,0,blend_radius_m)
    |   movel([0.454430, -1.439177, -2.533536, -0.739677, 1.570796, 2.025226],accel_mss,speed_ms,0,blend_radius_m)
    |   movel([0.453802, -1.438678, -2.533930, -0.739781, 1.570796, 2.024598],accel_mss,speed_ms,0,blend_radius_m)
    |   movel([0.453497, -1.437998, -2.534467, -0.739924, 1.570796, 2.024293],accel_mss,speed_ms,0,blend_radius_m)
    |   movel([0.453470, -1.437176, -2.535115, -0.740098, 1.570796, 2.024266],accel_mss,speed_ms,0,blend_radius_m)
    |   movel([0.453674, -1.436249, -2.535845, -0.740295, 1.570796, 2.024470],accel_mss,speed_ms,0,blend_radius_m)
    |   movel([0.454060, -1.435263, -2.536620, -0.740506, 1.570796, 2.024857],accel_mss,speed_ms,0,blend_radius_m)
    |   movel([0.454581, -1.434254, -2.537412, -0.740723, 1.570796, 2.025378],accel_mss,speed_ms,0,blend_radius_m)
    |   movel([0.455194, -1.433264, -2.538187, -0.740938, 1.570796, 2.025991],accel_mss,speed_ms,0,blend_radius_m)
    |   movel([0.456666, -1.431232, -2.539773, -0.741384, 1.570796, 2.027463],accel_mss,speed_ms,0,blend_radius_m)
    |   movel([0.458291, -1.429284, -2.541288, -0.741817, 1.570796, 2.029088],accel_mss,speed_ms,0,blend_radius_m)
    |   movel([0.461810, -1.425442, -2.544259, -0.742688, 1.570796, 2.032606],accel_mss,speed_ms,0,blend_radius_m)
    |   movel([0.459726, -1.420705, -2.547891, -0.743793, 1.570796, 2.030522],accel_mss,speed_ms,0,blend_radius_m)
    |   movel([0.457477, -1.416035, -2.551439, -0.744915, 1.570796, 2.028274],accel_mss,speed_ms,0,blend_radius_m)
    |   movel([0.455278, -1.411296, -2.555006, -0.746087, 1.570796, 2.026074],accel_mss,speed_ms,0,blend_radius_m)
    |   movel([0.454264, -1.408857, -2.556829, -0.746703, 1.570796, 2.025061],accel_mss,speed_ms,0,blend_radius_m)
    |   movel([0.453345, -1.406346, -2.558696, -0.747347, 1.570796, 2.024141],accel_mss,speed_ms,0,blend_radius_m)
    |   movel([0.452586, -1.403861, -2.560535, -0.747994, 1.570796, 2.023383],accel_mss,speed_ms,0,blend_radius_m)
    |   movel([0.451946, -1.401323, -2.562403, -0.748663, 1.570796, 2.022742],accel_mss,speed_ms,0,blend_radius_m)
    |   movel([0.450899, -1.396130, -2.566196, -0.750063, 1.570796, 2.021696],accel_mss,speed_ms,0,blend_radius_m)
    |   movel([0.449938, -1.390874, -2.569995, -0.751519, 1.570796, 2.020735],accel_mss,speed_ms,0,blend_radius_m)
    |   movel([0.448799, -1.385666, -2.573720, -0.753003, 1.570796, 2.019595],accel_mss,speed_ms,0,blend_radius_m)
    |   movel([0.446490, -1.387724, -2.572253, -0.752412, 1.570796, 2.017286],accel_mss,speed_ms,0,blend_radius_m)
    |   movel([0.444290, -1.389839, -2.570739, -0.751811, 1.570796, 2.015086],accel_mss,speed_ms,0,blend_radius_m)
    |   movel([0.442204, -1.392001, -2.569185, -0.751204, 1.570796, 2.013001],accel_mss,speed_ms,0,blend_radius_m)
    |   movel([0.440236, -1.394203, -2.567594, -0.750592, 1.570796, 2.011032],accel_mss,speed_ms,0,blend_radius_m)
    |   movel([0.438387, -1.396442, -2.565970, -0.749978, 1.570796, 2.009184],accel_mss,speed_ms,0,blend_radius_m)
    |   movel([0.436661, -1.398709, -2.564318, -0.749363, 1.570796, 2.007457],accel_mss,speed_ms,0,blend_radius_m)
    |   movel([0.435061, -1.401000, -2.562640, -0.748749, 1.570796, 2.005857],accel_mss,speed_ms,0,blend_radius_m)
    |   movel([0.433585, -1.403309, -2.560941, -0.748138, 1.570796, 2.004382],accel_mss,speed_ms,0,blend_radius_m)
    |   movel([0.432240, -1.405632, -2.559225, -0.747532, 1.570796, 2.003037],accel_mss,speed_ms,0,blend_radius_m)
    |   movel([0.431031, -1.407960, -2.557497, -0.746932, 1.570796, 2.001827],accel_mss,speed_ms,0,blend_radius_m)
    |   movel([0.429952, -1.410292, -2.555757, -0.746340, 1.570796, 2.000748],accel_mss,speed_ms,0,blend_radius_m)
    |   movel([0.429009, -1.412619, -2.554014, -0.745756, 1.570796, 1.999805],accel_mss,speed_ms,0,blend_radius_m)
    |   movel([0.428208, -1.414937, -2.552269, -0.745184, 1.570796, 1.999004],accel_mss,speed_ms,0,blend_radius_m)
    |   movel([0.427544, -1.417243, -2.550524, -0.744621, 1.570796, 1.998340],accel_mss,speed_ms,0,blend_radius_m)
    |   movel([0.427022, -1.419531, -2.548787, -0.744072, 1.570796, 1.997819],accel_mss,speed_ms,0,blend_radius_m)
    |   movel([0.426645, -1.421797, -2.547057, -0.743535, 1.570796, 1.997441],accel_mss,speed_ms,0,blend_radius_m)
    |   movel([0.426336, -1.425233, -2.544420, -0.742736, 1.570796, 1.997132],accel_mss,speed_ms,0,blend_radius_m)
    |   movel([0.426338, -1.428536, -2.541869, -0.741985, 1.570796, 1.997134],accel_mss,speed_ms,0,blend_radius_m)
    |   movel([0.426615, -1.431713, -2.539399, -0.741278, 1.570796, 1.997412],accel_mss,speed_ms,0,blend_radius_m)
    |   movel([0.427143, -1.434772, -2.537005, -0.740611, 1.570796, 1.997939],accel_mss,speed_ms,0,blend_radius_m)
    |   movel([0.427888, -1.437723, -2.534684, -0.739982, 1.570796, 1.998684],accel_mss,speed_ms,0,blend_radius_m)
    |   movel([0.428821, -1.440571, -2.532431, -0.739387, 1.570796, 1.999617],accel_mss,speed_ms,0,blend_radius_m)
    |   movel([0.429912, -1.443324, -2.530241, -0.738824, 1.570796, 2.000708],accel_mss,speed_ms,0,blend_radius_m)
    |   movel([0.431139, -1.445987, -2.528112, -0.738291, 1.570796, 2.001935],accel_mss,speed_ms,0,blend_radius_m)
    |   movel([0.433874, -1.451135, -2.523964, -0.737290, 1.570796, 2.004670],accel_mss,speed_ms,0,blend_radius_m)
    |   movel([0.436780, -1.456133, -2.519898, -0.736358, 1.570796, 2.007576],accel_mss,speed_ms,0,blend_radius_m)
    |   movel([0.438913, -1.460048, -2.516686, -0.735654, 1.570796, 2.009709],accel_mss,speed_ms,0,blend_radius_m)
    |   movel([0.439725, -1.461265, -2.515683, -0.735441, 1.570796, 2.010521],accel_mss,speed_ms,0,blend_radius_m)
    |   movel([0.441334, -1.463212, -2.514074, -0.735104, 1.570796, 2.012131],accel_mss,speed_ms,0,blend_radius_m)
    |   movel([0.441603, -1.463733, -2.513641, -0.735014, 1.570796, 2.012400],accel_mss,speed_ms,0,blend_radius_m)
    |   movel([0.441772, -1.464329, -2.513148, -0.734913, 1.570796, 2.012569],accel_mss,speed_ms,0,blend_radius_m)
    |   movel([0.441813, -1.465029, -2.512566, -0.734794, 1.570796, 2.012609],accel_mss,speed_ms,0,blend_radius_m)
    |   movel([0.441699, -1.465863, -2.511872, -0.734654, 1.570796, 2.012495],accel_mss,speed_ms,0,blend_radius_m)
    |   movel([0.441396, -1.466857, -2.511044, -0.734488, 1.570796, 2.012192],accel_mss,speed_ms,0,blend_radius_m)
    |   movel([0.440931, -1.467831, -2.510231, -0.734327, 1.570796, 2.011727],accel_mss,speed_ms,0,blend_radius_m)
    |   movel([0.440325, -1.468778, -2.509438, -0.734172, 1.570796, 2.011121],accel_mss,speed_ms,0,blend_radius_m)
    |   movel([0.439590, -1.469700, -2.508666, -0.734023, 1.570796, 2.010386],accel_mss,speed_ms,0,blend_radius_m)
    |   movel([0.438746, -1.470588, -2.507921, -0.733880, 1.570796, 2.009543],accel_mss,speed_ms,0,blend_radius_m)
    |   movel([0.436787, -1.472256, -2.506518, -0.733615, 1.570796, 2.007583],accel_mss,speed_ms,0,blend_radius_m)
    |   movel([0.435704, -1.473027, -2.505868, -0.733494, 1.570796, 2.006500],accel_mss,speed_ms,0,blend_radius_m)
    |   movel([0.433416, -1.474430, -2.504683, -0.733276, 1.570796, 2.004212],accel_mss,speed_ms,0,blend_radius_m)
    |   movel([0.431061, -1.475618, -2.503677, -0.733094, 1.570796, 2.001858],accel_mss,speed_ms,0,blend_radius_m)
    |   movel([0.428771, -1.476565, -2.502874, -0.732951, 1.570796, 1.999567],accel_mss,speed_ms,0,blend_radius_m)
    |   movel([0.426663, -1.477239, -2.502301, -0.732849, 1.570796, 1.997460],accel_mss,speed_ms,0,blend_radius_m)
    |   movel([0.423583, -1.477897, -2.501741, -0.732751, 1.570796, 1.994379],accel_mss,speed_ms,0,blend_radius_m)
    |   movel([0.422062, -1.478099, -2.501569, -0.732721, 1.570796, 1.992858],accel_mss,speed_ms,0,blend_radius_m)
    |   movel([0.420564, -1.478215, -2.501470, -0.732704, 1.570796, 1.991361],accel_mss,speed_ms,0,blend_radius_m)
    |   movel([0.417652, -1.478202, -2.501481, -0.732706, 1.570796, 1.988449],accel_mss,speed_ms,0,blend_radius_m)
    |   movel([0.414889, -1.477867, -2.501766, -0.732755, 1.570796, 1.985685],accel_mss,speed_ms,0,blend_radius_m)
    |   movel([0.412317, -1.477216, -2.502320, -0.732853, 1.570796, 1.983113],accel_mss,speed_ms,0,blend_radius_m)
    |   movel([0.409984, -1.476259, -2.503133, -0.732997, 1.570796, 1.980780],accel_mss,speed_ms,0,blend_radius_m)
    |   movel([0.408920, -1.475665, -2.503637, -0.733087, 1.570796, 1.979717],accel_mss,speed_ms,0,blend_radius_m)
    |   movel([0.407027, -1.474254, -2.504832, -0.733303, 1.570796, 1.977823],accel_mss,speed_ms,0,blend_radius_m)
    |   movel([0.406209, -1.473436, -2.505523, -0.733430, 1.570796, 1.977005],accel_mss,speed_ms,0,blend_radius_m)
    |   movel([0.405259, -1.472249, -2.506525, -0.733616, 1.570796, 1.976055],accel_mss,speed_ms,0,blend_radius_m)
    |   movel([0.404449, -1.470964, -2.507605, -0.733820, 1.570796, 1.975245],accel_mss,speed_ms,0,blend_radius_m)
    |   movel([0.403764, -1.469596, -2.508754, -0.734039, 1.570796, 1.974560],accel_mss,speed_ms,0,blend_radius_m)
    |   movel([0.403183, -1.468158, -2.509957, -0.734274, 1.570796, 1.973979],accel_mss,speed_ms,0,blend_radius_m)
    |   movel([0.402266, -1.465126, -2.512485, -0.734778, 1.570796, 1.973062],accel_mss,speed_ms,0,blend_radius_m)
    |   movel([0.401556, -1.461978, -2.515095, -0.735317, 1.570796, 1.972352],accel_mss,speed_ms,0,blend_radius_m)
    |   movel([0.400830, -1.457941, -2.518418, -0.736030, 1.570796, 1.971627],accel_mss,speed_ms,0,blend_radius_m)
    |   movel([0.400308, -1.453769, -2.521826, -0.736794, 1.570796, 1.971104],accel_mss,speed_ms,0,blend_radius_m)
    |   movel([0.400013, -1.449467, -2.525313, -0.737610, 1.570796, 1.970809],accel_mss,speed_ms,0,blend_radius_m)
    |   movel([0.399967, -1.445042, -2.528868, -0.738479, 1.570796, 1.970763],accel_mss,speed_ms,0,blend_radius_m)
    |   movel([0.400195, -1.440500, -2.532487, -0.739402, 1.570796, 1.970991],accel_mss,speed_ms,0,blend_radius_m)
    |   movel([0.400723, -1.435849, -2.536160, -0.740380, 1.570796, 1.971519],accel_mss,speed_ms,0,blend_radius_m)
    |   movel([0.401573, -1.431098, -2.539878, -0.741413, 1.570796, 1.972369],accel_mss,speed_ms,0,blend_radius_m)
    |   movel([0.402770, -1.426254, -2.543633, -0.742502, 1.570796, 1.973566],accel_mss,speed_ms,0,blend_radius_m)
    |   movel([0.403900, -1.422554, -2.546477, -0.743357, 1.570796, 1.974696],accel_mss,speed_ms,0,blend_radius_m)
    |   movel([0.405261, -1.418682, -2.549432, -0.744275, 1.570796, 1.976057],accel_mss,speed_ms,0,blend_radius_m)
    |   movel([0.406863, -1.414688, -2.552457, -0.745245, 1.570796, 1.977659],accel_mss,speed_ms,0,blend_radius_m)
    |   movel([0.408709, -1.410630, -2.555504, -0.746254, 1.570796, 1.979506],accel_mss,speed_ms,0,blend_radius_m)
    |   movel([0.410809, -1.406568, -2.558531, -0.747290, 1.570796, 1.981605],accel_mss,speed_ms,0,blend_radius_m)
    |   movel([0.413166, -1.402564, -2.561491, -0.748335, 1.570796, 1.983963],accel_mss,speed_ms,0,blend_radius_m)
    |   movel([0.415786, -1.398674, -2.564343, -0.749372, 1.570796, 1.986582],accel_mss,speed_ms,0,blend_radius_m)
    |   movel([0.417196, -1.396792, -2.565715, -0.749882, 1.570796, 1.987993],accel_mss,speed_ms,0,blend_radius_m)
    |   movel([0.418672, -1.394964, -2.567042, -0.750382, 1.570796, 1.989469],accel_mss,speed_ms,0,blend_radius_m)
    |   movel([0.421615, -1.391625, -2.569455, -0.751309, 1.570796, 1.992411],accel_mss,speed_ms,0,blend_radius_m)
    |   movel([0.424754, -1.388374, -2.571788, -0.752227, 1.570796, 1.995550],accel_mss,speed_ms,0,blend_radius_m)
    |   movel([0.428078, -1.385228, -2.574031, -0.753130, 1.570796, 1.998875],accel_mss,speed_ms,0,blend_radius_m)
    |   movel([0.431568, -1.382200, -2.576177, -0.754012, 1.570796, 2.002364],accel_mss,speed_ms,0,blend_radius_m)
    |   movel([0.435213, -1.379311, -2.578212, -0.754867, 1.570796, 2.006009],accel_mss,speed_ms,0,blend_radius_m)
    |   movel([0.438991, -1.376573, -2.580129, -0.755687, 1.570796, 2.009787],accel_mss,speed_ms,0,blend_radius_m)
    |   movel([0.442888, -1.374005, -2.581917, -0.756467, 1.570796, 2.013684],accel_mss,speed_ms,0,blend_radius_m)
    |   movel([0.446886, -1.371627, -2.583565, -0.757197, 1.570796, 2.017683],accel_mss,speed_ms,0,blend_radius_m)
    |   movel([0.447752, -1.362373, -2.589900, -0.760117, 1.570796, 2.018549],accel_mss,speed_ms,0,blend_radius_m)
    |   movel([0.448207, -1.357694, -2.593056, -0.761638, 1.570796, 2.019003],accel_mss,speed_ms,0,blend_radius_m)
    |   movel([0.448864, -1.352921, -2.596245, -0.763223, 1.570796, 2.019660],accel_mss,speed_ms,0,blend_radius_m)
    |   movel([0.449625, -1.349269, -2.598663, -0.764457, 1.570796, 2.020421],accel_mss,speed_ms,0,blend_radius_m)
    |   movel([0.450699, -1.345531, -2.601119, -0.765739, 1.570796, 2.021496],accel_mss,speed_ms,0,blend_radius_m)
    |   movel([0.452068, -1.341722, -2.603602, -0.767065, 1.570796, 2.022864],accel_mss,speed_ms,0,blend_radius_m)
    |   movel([0.453719, -1.337851, -2.606104, -0.768433, 1.570796, 2.024516],accel_mss,speed_ms,0,blend_radius_m)
    |   movel([0.455637, -1.333936, -2.608615, -0.769838, 1.570796, 2.026434],accel_mss,speed_ms,0,blend_radius_m)
    |   movel([0.457808, -1.329990, -2.611124, -0.771275, 1.570796, 2.028604],accel_mss,speed_ms,0,blend_radius_m)
    |   movel([0.460215, -1.326025, -2.613624, -0.772740, 1.570796, 2.031012],accel_mss,speed_ms,0,blend_radius_m)
    |   movel([0.462843, -1.322058, -2.616103, -0.774227, 1.570796, 2.033639],accel_mss,speed_ms,0,blend_radius_m)
    |   movel([0.465673, -1.318108, -2.618552, -0.775729, 1.570796, 2.036469],accel_mss,speed_ms,0,blend_radius_m)
    |   movel([0.468693, -1.314186, -2.620962, -0.777241, 1.570796, 2.039490],accel_mss,speed_ms,0,blend_radius_m)
    |   movel([0.471884, -1.310311, -2.623324, -0.778754, 1.570796, 2.042681],accel_mss,speed_ms,0,blend_radius_m)
    |   movel([0.475227, -1.306500, -2.625627, -0.780262, 1.570796, 2.046023],accel_mss,speed_ms,0,blend_radius_m)
    |   movel([0.478703, -1.302770, -2.627863, -0.781756, 1.570796, 2.049500],accel_mss,speed_ms,0,blend_radius_m)
    |   movel([0.482290, -1.299142, -2.630020, -0.783227, 1.570796, 2.053086],accel_mss,speed_ms,0,blend_radius_m)
    |   movel([0.485975, -1.295631, -2.632091, -0.784667, 1.570796, 2.056771],accel_mss,speed_ms,0,blend_radius_m)
    |   movel([0.489731, -1.292257, -2.634067, -0.786065, 1.570796, 2.060527],accel_mss,speed_ms,0,blend_radius_m)
    |   movel([0.496968, -1.286144, -2.637609, -0.788636, 1.570796, 2.067764],accel_mss,speed_ms,0,blend_radius_m)
    |   movel([0.500705, -1.283179, -2.639309, -0.789900, 1.570796, 2.071501],accel_mss,speed_ms,0,blend_radius_m)
    |   movel([0.504524, -1.280314, -2.640943, -0.791132, 1.570796, 2.075320],accel_mss,speed_ms,0,blend_radius_m)
    |   movel([0.508425, -1.277585, -2.642488, -0.792315, 1.570796, 2.079222],accel_mss,speed_ms,0,blend_radius_m)
    |   movel([0.512405, -1.275028, -2.643928, -0.793432, 1.570796, 2.083201],accel_mss,speed_ms,0,blend_radius_m)
    |   movel([0.516463, -1.272675, -2.645246, -0.794468, 1.570796, 2.087259],accel_mss,speed_ms,0,blend_radius_m)
    |   movel([0.520598, -1.270562, -2.646424, -0.795403, 1.570796, 2.091394],accel_mss,speed_ms,0,blend_radius_m)
    |   movel([0.525247, -1.268505, -2.647565, -0.796319, 1.570796, 2.096043],accel_mss,speed_ms,0,blend_radius_m)
    |   movel([0.529924, -1.266727, -2.648547, -0.797115, 1.570796, 2.100720],accel_mss,speed_ms,0,blend_radius_m)
    |   movel([0.534608, -1.265225, -2.649373, -0.797791, 1.570796, 2.105404],accel_mss,speed_ms,0,blend_radius_m)
    |   movel([0.539277, -1.263999, -2.650046, -0.798344, 1.570796, 2.110073],accel_mss,speed_ms,0,blend_radius_m)
    |   movel([0.543909, -1.263050, -2.650565, -0.798774, 1.570796, 2.114705],accel_mss,speed_ms,0,blend_radius_m)
    |   movel([0.548480, -1.262375, -2.650934, -0.799080, 1.570796, 2.119276],accel_mss,speed_ms,0,blend_radius_m)
    |   movel([0.552974, -1.261971, -2.651155, -0.799264, 1.570796, 2.123770],accel_mss,speed_ms,0,blend_radius_m)
    |   movel([0.557365, -1.261835, -2.651229, -0.799326, 1.570796, 2.128162],accel_mss,speed_ms,0,blend_radius_m)
    |   movel([0.561634, -1.261965, -2.651158, -0.799266, 1.570796, 2.132430],accel_mss,speed_ms,0,blend_radius_m)
    |   movel([0.565759, -1.262351, -2.650947, -0.799091, 1.570796, 2.136556],accel_mss,speed_ms,0,blend_radius_m)
    |   movel([0.569723, -1.262993, -2.650596, -0.798799, 1.570796, 2.140519],accel_mss,speed_ms,0,blend_radius_m)
    |   movel([0.573505, -1.263882, -2.650110, -0.798397, 1.570796, 2.144301],accel_mss,speed_ms,0,blend_radius_m)
    |   movel([0.577085, -1.265010, -2.649491, -0.797888, 1.570796, 2.147881],accel_mss,speed_ms,0,blend_radius_m)
    |   movel([0.580448, -1.266370, -2.648743, -0.797275, 1.570796, 2.151244],accel_mss,speed_ms,0,blend_radius_m)
    |   movel([0.583576, -1.267954, -2.647869, -0.796565, 1.570796, 2.154372],accel_mss,speed_ms,0,blend_radius_m)
    |   movel([0.586452, -1.269757, -2.646871, -0.795761, 1.570796, 2.157249],accel_mss,speed_ms,0,blend_radius_m)
    |   movel([0.589310, -1.271851, -2.645706, -0.794832, 1.570796, 2.160106],accel_mss,speed_ms,0,blend_radius_m)
    |   movel([0.592005, -1.274099, -2.644449, -0.793840, 1.570796, 2.162801],accel_mss,speed_ms,0,blend_radius_m)
    |   movel([0.594490, -1.276534, -2.643081, -0.792774, 1.570796, 2.165286],accel_mss,speed_ms,0,blend_radius_m)
    |   movel([0.596713, -1.279192, -2.641579, -0.791618, 1.570796, 2.167509],accel_mss,speed_ms,0,blend_radius_m)
    |   movel([0.598939, -1.282605, -2.639638, -0.790146, 1.570796, 2.169736],accel_mss,speed_ms,0,blend_radius_m)
    |   movel([0.600795, -1.286342, -2.637495, -0.788552, 1.570796, 2.171591],accel_mss,speed_ms,0,blend_radius_m)
    |   movel([0.602271, -1.290357, -2.635173, -0.786859, 1.570796, 2.173068],accel_mss,speed_ms,0,blend_radius_m)
    |   movel([0.603362, -1.294601, -2.632696, -0.785092, 1.570796, 2.174158],accel_mss,speed_ms,0,blend_radius_m)
    |   movel([0.604062, -1.299028, -2.630087, -0.783274, 1.570796, 2.174858],accel_mss,speed_ms,0,blend_radius_m)
    |   movel([0.604367, -1.303592, -2.627371, -0.781425, 1.570796, 2.175163],accel_mss,speed_ms,0,blend_radius_m)
    |   movel([0.604275, -1.308247, -2.624573, -0.779569, 1.570796, 2.175072],accel_mss,speed_ms,0,blend_radius_m)
    |   movel([0.603783, -1.312952, -2.621716, -0.777720, 1.570796, 2.174579],accel_mss,speed_ms,0,blend_radius_m)
    |   movel([0.602354, -1.322280, -2.615965, -0.774143, 1.570796, 2.173150],accel_mss,speed_ms,0,blend_radius_m)
    |   movel([0.601466, -1.326921, -2.613061, -0.772407, 1.570796, 2.172262],accel_mss,speed_ms,0,blend_radius_m)
    |   movel([0.600320, -1.331659, -2.610065, -0.770665, 1.570796, 2.171117],accel_mss,speed_ms,0,blend_radius_m)
    |   movel([0.598313, -1.339603, -2.604975, -0.767811, 1.570796, 2.169110],accel_mss,speed_ms,0,blend_radius_m)
    |   movel([0.597505, -1.343557, -2.602409, -0.766424, 1.570796, 2.168301],accel_mss,speed_ms,0,blend_radius_m)
    |   movel([0.596910, -1.347433, -2.599872, -0.765084, 1.570796, 2.167707],accel_mss,speed_ms,0,blend_radius_m)
    |   movel([0.596598, -1.351193, -2.597392, -0.763804, 1.570796, 2.167394],accel_mss,speed_ms,0,blend_radius_m)
    |   movel([0.596623, -1.354787, -2.595002, -0.762600, 1.570796, 2.167420],accel_mss,speed_ms,0,blend_radius_m)
    |   movel([0.597053, -1.358178, -2.592732, -0.761480, 1.570796, 2.167849],accel_mss,speed_ms,0,blend_radius_m)
    |   movel([0.597944, -1.361320, -2.590613, -0.760456, 1.570796, 2.168740],accel_mss,speed_ms,0,blend_radius_m)
    |   movel([0.598482, -1.362473, -2.589832, -0.760084, 1.570796, 2.169278],accel_mss,speed_ms,0,blend_radius_m)
    |   movel([0.599238, -1.363462, -2.589160, -0.759767, 1.570796, 2.170034],accel_mss,speed_ms,0,blend_radius_m)
    |   movel([0.599719, -1.363846, -2.588899, -0.759644, 1.570796, 2.170515],accel_mss,speed_ms,0,blend_radius_m)
    |   movel([0.600276, -1.364131, -2.588706, -0.759553, 1.570796, 2.171072],accel_mss,speed_ms,0,blend_radius_m)
    |   movel([0.600918, -1.364298, -2.588592, -0.759499, 1.570796, 2.171715],accel_mss,speed_ms,0,blend_radius_m)
    |   movel([0.601653, -1.364323, -2.588575, -0.759491, 1.570796, 2.172450],accel_mss,speed_ms,0,blend_radius_m)
    |   movel([0.602474, -1.364194, -2.588663, -0.759532, 1.570796, 2.173270],accel_mss,speed_ms,0,blend_radius_m)
    |   movel([0.603319, -1.363925, -2.588846, -0.759618, 1.570796, 2.174116],accel_mss,speed_ms,0,blend_radius_m)
    |   movel([0.605012, -1.363089, -2.589414, -0.759886, 1.570796, 2.175808],accel_mss,speed_ms,0,blend_radius_m)
    |   movel([0.606146, -1.362357, -2.589911, -0.760122, 1.570796, 2.176942],accel_mss,speed_ms,0,blend_radius_m)
    |   movel([0.607218, -1.361544, -2.590461, -0.760384, 1.570796, 2.178014],accel_mss,speed_ms,0,blend_radius_m)
    |   movel([0.609185, -1.359710, -2.591700, -0.760979, 1.570796, 2.179982],accel_mss,speed_ms,0,blend_radius_m)
    |   movel([0.610927, -1.357656, -2.593082, -0.761651, 1.570796, 2.181724],accel_mss,speed_ms,0,blend_radius_m)
    |   movel([0.612463, -1.355446, -2.594562, -0.762381, 1.570796, 2.183260],accel_mss,speed_ms,0,blend_radius_m)
    |   movel([0.613804, -1.353151, -2.596092, -0.763146, 1.570796, 2.184600],accel_mss,speed_ms,0,blend_radius_m)
    |   movel([0.614965, -1.350838, -2.597626, -0.763924, 1.570796, 2.185761],accel_mss,speed_ms,0,blend_radius_m)
    |   movel([0.615960, -1.348577, -2.599119, -0.764692, 1.570796, 2.186756],accel_mss,speed_ms,0,blend_radius_m)
    |   movel([0.617621, -1.344034, -2.602097, -0.766258, 1.570796, 2.188418],accel_mss,speed_ms,0,blend_radius_m)
    |   movel([0.618283, -1.341640, -2.603655, -0.767094, 1.570796, 2.189079],accel_mss,speed_ms,0,blend_radius_m)
    |   movel([0.618783, -1.339267, -2.605192, -0.767930, 1.570796, 2.189579],accel_mss,speed_ms,0,blend_radius_m)
    |   movel([0.619114, -1.336932, -2.606696, -0.768761, 1.570796, 2.189910],accel_mss,speed_ms,0,blend_radius_m)
    |   movel([0.619273, -1.334640, -2.608165, -0.769584, 1.570796, 2.190069],accel_mss,speed_ms,0,blend_radius_m)
    |   movel([0.619253, -1.332407, -2.609590, -0.770392, 1.570796, 2.190050],accel_mss,speed_ms,0,blend_radius_m)
    |   movel([0.619056, -1.330244, -2.610963, -0.771182, 1.570796, 2.189852],accel_mss,speed_ms,0,blend_radius_m)
    |   movel([0.618673, -1.328162, -2.612279, -0.771948, 1.570796, 2.189470],accel_mss,speed_ms,0,blend_radius_m)
    |   speed_ms = 0.005
    |   movel([0.618673, -1.318990, -2.608056, -0.785343, 1.570796, 2.189470],accel_mss,speed_ms,0,blend_radius_m)
    |   speed_ms = 0.040
    |   movel([0.608287, -1.336883, -2.596709, -0.778797, 1.570796, 2.179083],accel_mss,speed_ms,0,blend_radius_m)
    |   speed_ms = 0.005
    |   movel([0.608287, -1.345938, -2.600853, -0.765598, 1.570796, 2.179083],accel_mss,speed_ms,0,blend_radius_m)
    |   speed_ms = 0.025
    |   movel([0.607618, -1.343589, -2.602388, -0.766412, 1.570796, 2.178415],accel_mss,speed_ms,0,blend_radius_m)
    |   movel([0.606621, -1.341427, -2.603794, -0.767169, 1.570796, 2.177417],accel_mss,speed_ms,0,blend_radius_m)
    |   movel([0.605939, -1.340487, -2.604403, -0.767499, 1.570796, 2.176735],accel_mss,speed_ms,0,blend_radius_m)
    |   movel([0.605103, -1.339682, -2.604923, -0.767783, 1.570796, 2.175900],accel_mss,speed_ms,0,blend_radius_m)
    |   movel([0.604092, -1.339042, -2.605337, -0.768010, 1.570796, 2.174888],accel_mss,speed_ms,0,blend_radius_m)
    |   movel([0.602882, -1.338593, -2.605627, -0.768169, 1.570796, 2.173679],accel_mss,speed_ms,0,blend_radius_m)
    |   speed_ms = 0.005
    |   movel([0.602882, -1.329489, -2.601450, -0.781450, 1.570796, 2.173679],accel_mss,speed_ms,0,blend_radius_m)
    |   speed_ms = 0.040
    |   movel([0.608939, -1.326488, -2.603353, -0.782548, 1.570796, 2.179736],accel_mss,speed_ms,0,blend_radius_m)
    |   speed_ms = 0.005
    |   movel([0.608939, -1.335612, -2.607543, -0.769234, 1.570796, 2.179736],accel_mss,speed_ms,0,blend_radius_m)
    |   speed_ms = 0.025
    |   movel([0.610243, -1.333197, -2.609086, -0.770105, 1.570796, 2.181039],accel_mss,speed_ms,0,blend_radius_m)
    |   movel([0.611107, -1.330823, -2.610596, -0.770970, 1.570796, 2.181903],accel_mss,speed_ms,0,blend_radius_m)
    |   movel([0.611540, -1.328533, -2.612045, -0.771811, 1.570796, 2.182336],accel_mss,speed_ms,0,blend_radius_m)
    |   movel([0.611538, -1.326385, -2.613398, -0.772606, 1.570796, 2.182334],accel_mss,speed_ms,0,blend_radius_m)
    |   movel([0.611105, -1.324430, -2.614624, -0.773336, 1.570796, 2.181902],accel_mss,speed_ms,0,blend_radius_m)
    |   movel([0.610245, -1.322725, -2.615688, -0.773976, 1.570796, 2.181041],accel_mss,speed_ms,0,blend_radius_m)
    |   movel([0.608961, -1.321322, -2.616562, -0.774506, 1.570796, 2.179757],accel_mss,speed_ms,0,blend_radius_m)
    |   movel([0.608159, -1.320752, -2.616916, -0.774722, 1.570796, 2.178955],accel_mss,speed_ms,0,blend_radius_m)
    |   movel([0.607255, -1.320275, -2.617211, -0.774903, 1.570796, 2.178051],accel_mss,speed_ms,0,blend_radius_m)
    |   speed_ms = 0.005
    |   movel([0.607255, -1.311053, -2.612952, -0.788384, 1.570796, 2.178051],accel_mss,speed_ms,0,blend_radius_m)
    |   speed_ms = 0.040
    |   movel([0.613864, -1.309274, -2.614039, -0.789077, 1.570796, 2.184660],accel_mss,speed_ms,0,blend_radius_m)
    |   speed_ms = 0.005
    |   movel([0.613864, -1.318507, -2.618305, -0.775576, 1.570796, 2.184660],accel_mss,speed_ms,0,blend_radius_m)
    |   speed_ms = 0.025
    |   movel([0.614362, -1.317270, -2.619068, -0.776050, 1.570796, 2.185158],accel_mss,speed_ms,0,blend_radius_m)
    |   movel([0.614733, -1.316020, -2.619838, -0.776531, 1.570796, 2.185530],accel_mss,speed_ms,0,blend_radius_m)
    |   movel([0.615108, -1.313519, -2.621370, -0.777500, 1.570796, 2.185904],accel_mss,speed_ms,0,blend_radius_m)
    |   movel([0.615013, -1.311091, -2.622850, -0.778448, 1.570796, 2.185809],accel_mss,speed_ms,0,blend_radius_m)
    |   movel([0.614473, -1.308828, -2.624222, -0.779339, 1.570796, 2.185269],accel_mss,speed_ms,0,blend_radius_m)
    |   movel([0.613517, -1.306811, -2.625439, -0.780138, 1.570796, 2.184314],accel_mss,speed_ms,0,blend_radius_m)
    |   movel([0.612179, -1.305135, -2.626447, -0.780807, 1.570796, 2.182975],accel_mss,speed_ms,0,blend_radius_m)
    |   movel([0.611372, -1.304453, -2.626856, -0.781080, 1.570796, 2.182168],accel_mss,speed_ms,0,blend_radius_m)
    |   movel([0.609512, -1.303452, -2.627455, -0.781482, 1.570796, 2.180308],accel_mss,speed_ms,0,blend_radius_m)
    |   movel([0.608466, -1.303155, -2.627633, -0.781601, 1.570796, 2.179262],accel_mss,speed_ms,0,blend_radius_m)
    |   speed_ms = 0.005
    |   movel([0.608466, -1.293828, -2.623296, -0.795265, 1.570796, 2.179262],accel_mss,speed_ms,0,blend_radius_m)
    |   speed_ms = 0.040
    |   movel([0.617198, -1.292574, -2.624034, -0.795781, 1.570796, 2.187994],accel_mss,speed_ms,0,blend_radius_m)
    |   speed_ms = 0.005
    |   movel([0.617198, -1.301908, -2.628377, -0.782104, 1.570796, 2.187994],accel_mss,speed_ms,0,blend_radius_m)
    |   speed_ms = 0.025
    |   movel([0.617312, -1.299065, -2.630065, -0.783259, 1.570796, 2.188108],accel_mss,speed_ms,0,blend_radius_m)
    |   movel([0.617008, -1.296386, -2.631647, -0.784356, 1.570796, 2.187804],accel_mss,speed_ms,0,blend_radius_m)
    |   movel([0.616278, -1.293946, -2.633079, -0.785363, 1.570796, 2.187075],accel_mss,speed_ms,0,blend_radius_m)
    |   movel([0.615115, -1.291804, -2.634331, -0.786254, 1.570796, 2.185912],accel_mss,speed_ms,0,blend_radius_m)
    |   movel([0.613512, -1.290032, -2.635361, -0.786996, 1.570796, 2.184309],accel_mss,speed_ms,0,blend_radius_m)
    |   movel([0.612545, -1.289304, -2.635784, -0.787301, 1.570796, 2.183341],accel_mss,speed_ms,0,blend_radius_m)
    |   movel([0.611467, -1.288695, -2.636136, -0.787558, 1.570796, 2.182263],accel_mss,speed_ms,0,blend_radius_m)
    |   movel([0.610275, -1.288211, -2.636417, -0.787762, 1.570796, 2.181072],accel_mss,speed_ms,0,blend_radius_m)
    |   movel([0.608969, -1.287860, -2.636619, -0.787910, 1.570796, 2.179766],accel_mss,speed_ms,0,blend_radius_m)
    |   movel([0.607554, -1.287651, -2.636740, -0.787998, 1.570796, 2.178350],accel_mss,speed_ms,0,blend_radius_m)
    |   movel([0.606026, -1.287590, -2.636775, -0.788024, 1.570796, 2.176822],accel_mss,speed_ms,0,blend_radius_m)
    |   speed_ms = 0.005
    |   movel([0.606026, -1.278173, -2.632367, -0.801848, 1.570796, 2.176822],accel_mss,speed_ms,0,blend_radius_m)
    |   speed_ms = 0.040
    |   movel([0.616189, -1.275408, -2.633938, -0.803043, 1.570796, 2.186985],accel_mss,speed_ms,0,blend_radius_m)
    |   speed_ms = 0.005
    |   movel([0.616189, -1.284841, -2.638358, -0.789190, 1.570796, 2.186985],accel_mss,speed_ms,0,blend_radius_m)
    |   speed_ms = 0.025
    |   movel([0.616786, -1.282923, -2.639456, -0.790010, 1.570796, 2.187583],accel_mss,speed_ms,0,blend_radius_m)
    |   movel([0.617111, -1.281060, -2.640519, -0.790811, 1.570796, 2.187908],accel_mss,speed_ms,0,blend_radius_m)
    |   movel([0.617157, -1.279285, -2.641527, -0.791577, 1.570796, 2.187953],accel_mss,speed_ms,0,blend_radius_m)
    |   movel([0.616917, -1.277640, -2.642458, -0.792292, 1.570796, 2.187714],accel_mss,speed_ms,0,blend_radius_m)
    |   movel([0.616271, -1.275858, -2.643462, -0.793069, 1.570796, 2.187067],accel_mss,speed_ms,0,blend_radius_m)
    |   movel([0.615324, -1.274279, -2.644349, -0.793761, 1.570796, 2.186120],accel_mss,speed_ms,0,blend_radius_m)
    |   movel([0.613936, -1.272635, -2.645269, -0.794486, 1.570796, 2.184732],accel_mss,speed_ms,0,blend_radius_m)
    |   movel([0.612259, -1.271257, -2.646037, -0.795095, 1.570796, 2.183056],accel_mss,speed_ms,0,blend_radius_m)
    |   movel([0.610290, -1.270206, -2.646622, -0.795562, 1.570796, 2.181086],accel_mss,speed_ms,0,blend_radius_m)
    |   movel([0.608020, -1.269545, -2.646989, -0.795856, 1.570796, 2.178817],accel_mss,speed_ms,0,blend_radius_m)
    |   movel([0.605453, -1.269343, -2.647101, -0.795946, 1.570796, 2.176250],accel_mss,speed_ms,0,blend_radius_m)
    |   movel([0.604079, -1.269427, -2.647054, -0.795908, 1.570796, 2.174875],accel_mss,speed_ms,0,blend_radius_m)
    |   movel([0.601207, -1.269986, -2.646744, -0.795659, 1.570796, 2.172003],accel_mss,speed_ms,0,blend_radius_m)
    |   movel([0.599734, -1.270459, -2.646481, -0.795449, 1.570796, 2.170531],accel_mss,speed_ms,0,blend_radius_m)
    |   movel([0.598254, -1.271070, -2.646141, -0.795178, 1.570796, 2.169050],accel_mss,speed_ms,0,blend_radius_m)
    |   movel([0.596777, -1.271817, -2.645725, -0.794847, 1.570796, 2.167573],accel_mss,speed_ms,0,blend_radius_m)
    |   speed_ms = 0.005
    |   movel([0.596777, -1.262313, -2.641245, -0.808830, 1.570796, 2.167573],accel_mss,speed_ms,0,blend_radius_m)
    |   speed_ms = 0.040
    |   movel([0.610162, -1.255273, -2.645088, -0.812028, 1.570796, 2.180958],accel_mss,speed_ms,0,blend_radius_m)
    |   speed_ms = 0.005
    |   movel([0.610162, -1.264814, -2.649599, -0.797976, 1.570796, 2.180958],accel_mss,speed_ms,0,blend_radius_m)
    |   speed_ms = 0.025
    |   movel([0.608223, -1.262806, -2.650699, -0.798885, 1.570796, 2.179019],accel_mss,speed_ms,0,blend_radius_m)
    |   movel([0.605896, -1.261103, -2.651627, -0.799658, 1.570796, 2.176692],accel_mss,speed_ms,0,blend_radius_m)
    |   movel([0.603204, -1.259803, -2.652334, -0.800252, 1.570796, 2.174000],accel_mss,speed_ms,0,blend_radius_m)
    |   movel([0.601731, -1.259331, -2.652590, -0.800468, 1.570796, 2.172527],accel_mss,speed_ms,0,blend_radius_m)
    |   movel([0.600177, -1.258994, -2.652773, -0.800622, 1.570796, 2.170973],accel_mss,speed_ms,0,blend_radius_m)
    |   movel([0.598548, -1.258803, -2.652876, -0.800710, 1.570796, 2.169344],accel_mss,speed_ms,0,blend_radius_m)
    |   movel([0.596850, -1.258769, -2.652894, -0.800725, 1.570796, 2.167646],accel_mss,speed_ms,0,blend_radius_m)
    |   movel([0.595084, -1.258904, -2.652822, -0.800664, 1.570796, 2.165881],accel_mss,speed_ms,0,blend_radius_m)
    |   movel([0.593255, -1.259219, -2.652651, -0.800519, 1.570796, 2.164052],accel_mss,speed_ms,0,blend_radius_m)
    |   movel([0.591368, -1.259721, -2.652378, -0.800289, 1.570796, 2.162164],accel_mss,speed_ms,0,blend_radius_m)
    |   movel([0.589429, -1.260425, -2.651996, -0.799968, 1.570796, 2.160226],accel_mss,speed_ms,0,blend_radius_m)
    |   movel([0.587443, -1.261337, -2.651500, -0.799552, 1.570796, 2.158239],accel_mss,speed_ms,0,blend_radius_m)
    |   movel([0.585414, -1.262471, -2.650882, -0.799036, 1.570796, 2.156210],accel_mss,speed_ms,0,blend_radius_m)
    |   speed_ms = 0.005
    |   movel([0.585414, -1.252918, -2.646359, -0.813111, 1.570796, 2.156210],accel_mss,speed_ms,0,blend_radius_m)
    |   speed_ms = 0.040
    |   movel([0.598369, -1.242369, -2.651976, -0.818045, 1.570796, 2.169165],accel_mss,speed_ms,0,blend_radius_m)
    |   speed_ms = 0.005
    |   movel([0.598369, -1.251973, -2.656546, -0.803869, 1.570796, 2.169165],accel_mss,speed_ms,0,blend_radius_m)
    |   speed_ms = 0.025
    |   movel([0.597272, -1.251063, -2.657031, -0.804295, 1.570796, 2.168068],accel_mss,speed_ms,0,blend_radius_m)
    |   movel([0.596023, -1.250312, -2.657430, -0.804646, 1.570796, 2.166820],accel_mss,speed_ms,0,blend_radius_m)
    |   movel([0.594635, -1.249734, -2.657737, -0.804918, 1.570796, 2.165431],accel_mss,speed_ms,0,blend_radius_m)
    |   movel([0.593122, -1.249325, -2.657954, -0.805110, 1.570796, 2.163918],accel_mss,speed_ms,0,blend_radius_m)
    |   movel([0.591496, -1.249090, -2.658079, -0.805220, 1.570796, 2.162292],accel_mss,speed_ms,0,blend_radius_m)
    |   movel([0.589773, -1.249035, -2.658108, -0.805246, 1.570796, 2.160569],accel_mss,speed_ms,0,blend_radius_m)
    |   movel([0.587971, -1.249158, -2.658042, -0.805188, 1.570796, 2.158767],accel_mss,speed_ms,0,blend_radius_m)
    |   movel([0.586097, -1.249465, -2.657880, -0.805044, 1.570796, 2.156894],accel_mss,speed_ms,0,blend_radius_m)
    |   movel([0.584175, -1.249956, -2.657620, -0.804814, 1.570796, 2.154971],accel_mss,speed_ms,0,blend_radius_m)
    |   movel([0.582222, -1.250621, -2.657266, -0.804502, 1.570796, 2.153019],accel_mss,speed_ms,0,blend_radius_m)
    |   movel([0.580260, -1.251450, -2.656825, -0.804114, 1.570796, 2.151056],accel_mss,speed_ms,0,blend_radius_m)
    |   movel([0.578304, -1.252435, -2.656300, -0.803654, 1.570796, 2.149100],accel_mss,speed_ms,0,blend_radius_m)
    |   movel([0.576372, -1.253561, -2.655698, -0.803130, 1.570796, 2.147169],accel_mss,speed_ms,0,blend_radius_m)
